// ---- DUTs/IO/Boxes/ER1008_78E8D3DD.TcDUT
{attribute 'GeneratedUsingTerminal: ER1008-0001-0016'}
{attribute addProperty BoxType "ER1008-0001-0016"}
{attribute addProperty Description "ER1008-0001 8 Ch. Dig. Input 24V, 3ms, M8"}
{attribute addProperty Physics "YY"}
{attribute addProperty Id "Channel_1AT %I*Channel_830843C11Channel_2AT %I*Channel_830843C11Channel_3AT %I*Channel_830843C11Channel_4AT %I*Channel_830843C11Channel_5AT %I*Channel_830843C11Channel_6AT %I*Channel_830843C11Channel_7AT %I*Channel_830843C11Channel_8AT %I*Channel_830843C11WcStateAT %I*WcState_9091E0EB2InfoDataAT %I*InfoData_6F19DB2B2"}
{attribute addProperty CRC "2028524509"}
{attribute addProperty Size "12"}
TYPE ER1008_78E8D3DD EXTENDS EtcSlaveBoxBase_77A0E4A7 :
STRUCT
	{attribute addProperty Name "Channel_1"}
	Channel_1 : Channel_830843C1;
	{attribute addProperty Name "Channel_2"}
	Channel_2 : Channel_830843C1;
	{attribute addProperty Name "Channel_3"}
	Channel_3 : Channel_830843C1;
	{attribute addProperty Name "Channel_4"}
	Channel_4 : Channel_830843C1;
	{attribute addProperty Name "Channel_5"}
	Channel_5 : Channel_830843C1;
	{attribute addProperty Name "Channel_6"}
	Channel_6 : Channel_830843C1;
	{attribute addProperty Name "Channel_7"}
	Channel_7 : Channel_830843C1;
	{attribute addProperty Name "Channel_8"}
	Channel_8 : Channel_830843C1;
	{attribute addProperty Name "WcState"}
	WcState : WcState_9091E0EB;
	{attribute addProperty Name "InfoData"}
	InfoData : InfoData_6F19DB2B;
END_STRUCT
END_TYPE

// ---- DUTs/IO/Boxes/ER1018_78E8D3DD.TcDUT
{attribute 'GeneratedUsingTerminal: ER1018-0001-0018'}
{attribute addProperty BoxType "ER1018-0001-0018"}
{attribute addProperty Description "ER1018-0001 8 Ch. Dig. Input 24V, 10µs, M8"}
{attribute addProperty Physics "YY"}
{attribute addProperty Id "Channel_1AT %I*Channel_830843C11Channel_2AT %I*Channel_830843C11Channel_3AT %I*Channel_830843C11Channel_4AT %I*Channel_830843C11Channel_5AT %I*Channel_830843C11Channel_6AT %I*Channel_830843C11Channel_7AT %I*Channel_830843C11Channel_8AT %I*Channel_830843C11WcStateAT %I*WcState_9091E0EB2InfoDataAT %I*InfoData_6F19DB2B2"}
{attribute addProperty CRC "2028524509"}
{attribute addProperty Size "12"}
TYPE ER1018_78E8D3DD EXTENDS EtcSlaveBoxBase_77A0E4A7 :
STRUCT
	{attribute addProperty Name "Channel_1"}
	Channel_1 : Channel_830843C1;
	{attribute addProperty Name "Channel_2"}
	Channel_2 : Channel_830843C1;
	{attribute addProperty Name "Channel_3"}
	Channel_3 : Channel_830843C1;
	{attribute addProperty Name "Channel_4"}
	Channel_4 : Channel_830843C1;
	{attribute addProperty Name "Channel_5"}
	Channel_5 : Channel_830843C1;
	{attribute addProperty Name "Channel_6"}
	Channel_6 : Channel_830843C1;
	{attribute addProperty Name "Channel_7"}
	Channel_7 : Channel_830843C1;
	{attribute addProperty Name "Channel_8"}
	Channel_8 : Channel_830843C1;
	{attribute addProperty Name "WcState"}
	WcState : WcState_9091E0EB;
	{attribute addProperty Name "InfoData"}
	InfoData : InfoData_6F19DB2B;
END_STRUCT
END_TYPE

// ---- DUTs/IO/Boxes/ER1098_78E8D3DD.TcDUT
{attribute 'GeneratedUsingTerminal: ER1098-0001-0017'}
{attribute addProperty BoxType "ER1098-0001-0017"}
{attribute addProperty Description "ER1098-0001 8 Ch. Dig. Input 24V, 10us, M8, negative"}
{attribute addProperty Physics "YY"}
{attribute addProperty Id "Channel_1AT %I*Channel_830843C11Channel_2AT %I*Channel_830843C11Channel_3AT %I*Channel_830843C11Channel_4AT %I*Channel_830843C11Channel_5AT %I*Channel_830843C11Channel_6AT %I*Channel_830843C11Channel_7AT %I*Channel_830843C11Channel_8AT %I*Channel_830843C11WcStateAT %I*WcState_9091E0EB2InfoDataAT %I*InfoData_6F19DB2B2"}
{attribute addProperty CRC "2028524509"}
{attribute addProperty Size "12"}
TYPE ER1098_78E8D3DD EXTENDS EtcSlaveBoxBase_77A0E4A7 :
STRUCT
	{attribute addProperty Name "Channel_1"}
	Channel_1 : Channel_830843C1;
	{attribute addProperty Name "Channel_2"}
	Channel_2 : Channel_830843C1;
	{attribute addProperty Name "Channel_3"}
	Channel_3 : Channel_830843C1;
	{attribute addProperty Name "Channel_4"}
	Channel_4 : Channel_830843C1;
	{attribute addProperty Name "Channel_5"}
	Channel_5 : Channel_830843C1;
	{attribute addProperty Name "Channel_6"}
	Channel_6 : Channel_830843C1;
	{attribute addProperty Name "Channel_7"}
	Channel_7 : Channel_830843C1;
	{attribute addProperty Name "Channel_8"}
	Channel_8 : Channel_830843C1;
	{attribute addProperty Name "WcState"}
	WcState : WcState_9091E0EB;
	{attribute addProperty Name "InfoData"}
	InfoData : InfoData_6F19DB2B;
END_STRUCT
END_TYPE

// ---- DUTs/IO/Boxes/ER1258_58F475DD.TcDUT
{attribute 'GeneratedUsingTerminal: ER1258-0001-0019'}
{attribute addProperty BoxType "ER1258-0001-0019"}
{attribute addProperty Description "ER1258-0001 8 Ch. Dig. Input 24V, 10µs, DC Latch, M8"}
{attribute addProperty Physics "YY"}
{attribute addProperty Id "Channel_1AT %I*Channel_830843C11Channel_2AT %I*Channel_830843C11Channel_3AT %I*Channel_830843C11Channel_4AT %I*Channel_830843C11Channel_5AT %I*Channel_830843C11Channel_6AT %I*Channel_830843C11Channel_7AT %I*Channel_830843C11Channel_8AT %I*Channel_830843C11LatchAT %I*Latch_8E41329534WcStateAT %I*WcState_B516A2644InfoDataAT %I*InfoData_A7436BC610"}
{attribute addProperty CRC "1492415965"}
{attribute addProperty Size "56"}
TYPE ER1258_58F475DD EXTENDS EtcSlaveBoxBase_77A0E4A7 :
STRUCT
	{attribute addProperty Name "Channel_1"}
	Channel_1 : Channel_830843C1;
	{attribute addProperty Name "Channel_2"}
	Channel_2 : Channel_830843C1;
	{attribute addProperty Name "Channel_3"}
	Channel_3 : Channel_830843C1;
	{attribute addProperty Name "Channel_4"}
	Channel_4 : Channel_830843C1;
	{attribute addProperty Name "Channel_5"}
	Channel_5 : Channel_830843C1;
	{attribute addProperty Name "Channel_6"}
	Channel_6 : Channel_830843C1;
	{attribute addProperty Name "Channel_7"}
	Channel_7 : Channel_830843C1;
	{attribute addProperty Name "Channel_8"}
	Channel_8 : Channel_830843C1;
	{attribute addProperty Name "Latch"}
	Latch : Latch_8E413295;
	{attribute addProperty Name "WcState"}
	WcState : WcState_B516A264;
	{attribute addProperty Name "InfoData"}
	InfoData : InfoData_A7436BC6;
END_STRUCT
END_TYPE

// ---- DUTs/IO/Boxes/ER1518_CC442588.TcDUT
{attribute 'GeneratedUsingTerminal: ER1518-0002-0018'}
{attribute addProperty BoxType "ER1518-0002-0018"}
{attribute addProperty Description "ER1518-0002 8 Ch.digital multi-function input"}
{attribute addProperty Physics "YY"}
{attribute addProperty Id "CNT_Input_Channel_1AT %I*CNT_Input_Channel_FF10BD3C11CNT_Input_Channel_2AT %I*CNT_Input_Channel_FF10BD3C11DIG_InputsAT %I*DIG_Inputs_CAFF60048DIG_Inputs_DeviceAT %I*DIG_Inputs_Device_1F4E72EB5CNT_Output_Channel_1AT %Q*CNT_Output_Channel_550BB6DF6CNT_Output_Channel_2AT %Q*CNT_Output_Channel_550BB6DF6WcStateAT %I*WcState_9091E0EB2InfoDataAT %I*InfoData_32EB74EA10"}
{attribute addProperty CRC "3427018120"}
{attribute addProperty Size "59"}
TYPE ER1518_CC442588 EXTENDS EtcSlaveBoxBase_77A0E4A7 :
STRUCT
	{attribute addProperty Name "CNT_Input_Channel_1"}
	CNT_Input_Channel_1 : CNT_Input_Channel_FF10BD3C;
	{attribute addProperty Name "CNT_Input_Channel_2"}
	CNT_Input_Channel_2 : CNT_Input_Channel_FF10BD3C;
	{attribute addProperty Name "DIG_Inputs"}
	DIG_Inputs : DIG_Inputs_CAFF6004;
	{attribute addProperty Name "DIG_Inputs_Device"}
	DIG_Inputs_Device : DIG_Inputs_Device_1F4E72EB;
	{attribute addProperty Name "CNT_Output_Channel_1"}
	CNT_Output_Channel_1 : CNT_Output_Channel_550BB6DF;
	{attribute addProperty Name "CNT_Output_Channel_2"}
	CNT_Output_Channel_2 : CNT_Output_Channel_550BB6DF;
	{attribute addProperty Name "WcState"}
	WcState : WcState_9091E0EB;
	{attribute addProperty Name "InfoData"}
	InfoData : InfoData_32EB74EA;
END_STRUCT
END_TYPE

// ---- DUTs/IO/Boxes/ER1809_32157CFD.TcDUT
{attribute 'GeneratedUsingTerminal: ER1809-0021-0017'}
{attribute addProperty BoxType "ER1809-0021-0017"}
{attribute addProperty Description "ER1809-0021 16 Ch. Dig. Input 24V, 3ms, M8"}
{attribute addProperty Physics "YY"}
{attribute addProperty Id "Channel_1AT %I*Channel_830843C11Channel_2AT %I*Channel_830843C11Channel_3AT %I*Channel_830843C11Channel_4AT %I*Channel_830843C11Channel_5AT %I*Channel_830843C11Channel_6AT %I*Channel_830843C11Channel_7AT %I*Channel_830843C11Channel_8AT %I*Channel_830843C11Channel_9AT %I*Channel_830843C11Channel_10AT %I*Channel_830843C11Channel_11AT %I*Channel_830843C11Channel_12AT %I*Channel_830843C11Channel_13AT %I*Channel_830843C11Channel_14AT %I*Channel_830843C11Channel_15AT %I*Channel_830843C11Channel_16AT %I*Channel_830843C11WcStateAT %I*WcState_9091E0EB2InfoDataAT %I*InfoData_6F19DB2B2"}
{attribute addProperty CRC "840269053"}
{attribute addProperty Size "20"}
TYPE ER1809_32157CFD EXTENDS EtcSlaveBoxBase_77A0E4A7 :
STRUCT
	{attribute addProperty Name "Channel_1"}
	Channel_1 : Channel_830843C1;
	{attribute addProperty Name "Channel_2"}
	Channel_2 : Channel_830843C1;
	{attribute addProperty Name "Channel_3"}
	Channel_3 : Channel_830843C1;
	{attribute addProperty Name "Channel_4"}
	Channel_4 : Channel_830843C1;
	{attribute addProperty Name "Channel_5"}
	Channel_5 : Channel_830843C1;
	{attribute addProperty Name "Channel_6"}
	Channel_6 : Channel_830843C1;
	{attribute addProperty Name "Channel_7"}
	Channel_7 : Channel_830843C1;
	{attribute addProperty Name "Channel_8"}
	Channel_8 : Channel_830843C1;
	{attribute addProperty Name "Channel_9"}
	Channel_9 : Channel_830843C1;
	{attribute addProperty Name "Channel_10"}
	Channel_10 : Channel_830843C1;
	{attribute addProperty Name "Channel_11"}
	Channel_11 : Channel_830843C1;
	{attribute addProperty Name "Channel_12"}
	Channel_12 : Channel_830843C1;
	{attribute addProperty Name "Channel_13"}
	Channel_13 : Channel_830843C1;
	{attribute addProperty Name "Channel_14"}
	Channel_14 : Channel_830843C1;
	{attribute addProperty Name "Channel_15"}
	Channel_15 : Channel_830843C1;
	{attribute addProperty Name "Channel_16"}
	Channel_16 : Channel_830843C1;
	{attribute addProperty Name "WcState"}
	WcState : WcState_9091E0EB;
	{attribute addProperty Name "InfoData"}
	InfoData : InfoData_6F19DB2B;
END_STRUCT
END_TYPE

// ---- DUTs/IO/Boxes/ER1819_32157CFD.TcDUT
{attribute 'GeneratedUsingTerminal: ER1819-0021-0017'}
{attribute addProperty BoxType "ER1819-0021-0017"}
{attribute addProperty Description "ER1819-0021 16 Ch. Dig. Input 24V, 10µs, M8"}
{attribute addProperty Physics "YY"}
{attribute addProperty Id "Channel_1AT %I*Channel_830843C11Channel_2AT %I*Channel_830843C11Channel_3AT %I*Channel_830843C11Channel_4AT %I*Channel_830843C11Channel_5AT %I*Channel_830843C11Channel_6AT %I*Channel_830843C11Channel_7AT %I*Channel_830843C11Channel_8AT %I*Channel_830843C11Channel_9AT %I*Channel_830843C11Channel_10AT %I*Channel_830843C11Channel_11AT %I*Channel_830843C11Channel_12AT %I*Channel_830843C11Channel_13AT %I*Channel_830843C11Channel_14AT %I*Channel_830843C11Channel_15AT %I*Channel_830843C11Channel_16AT %I*Channel_830843C11WcStateAT %I*WcState_9091E0EB2InfoDataAT %I*InfoData_6F19DB2B2"}
{attribute addProperty CRC "840269053"}
{attribute addProperty Size "20"}
TYPE ER1819_32157CFD EXTENDS EtcSlaveBoxBase_77A0E4A7 :
STRUCT
	{attribute addProperty Name "Channel_1"}
	Channel_1 : Channel_830843C1;
	{attribute addProperty Name "Channel_2"}
	Channel_2 : Channel_830843C1;
	{attribute addProperty Name "Channel_3"}
	Channel_3 : Channel_830843C1;
	{attribute addProperty Name "Channel_4"}
	Channel_4 : Channel_830843C1;
	{attribute addProperty Name "Channel_5"}
	Channel_5 : Channel_830843C1;
	{attribute addProperty Name "Channel_6"}
	Channel_6 : Channel_830843C1;
	{attribute addProperty Name "Channel_7"}
	Channel_7 : Channel_830843C1;
	{attribute addProperty Name "Channel_8"}
	Channel_8 : Channel_830843C1;
	{attribute addProperty Name "Channel_9"}
	Channel_9 : Channel_830843C1;
	{attribute addProperty Name "Channel_10"}
	Channel_10 : Channel_830843C1;
	{attribute addProperty Name "Channel_11"}
	Channel_11 : Channel_830843C1;
	{attribute addProperty Name "Channel_12"}
	Channel_12 : Channel_830843C1;
	{attribute addProperty Name "Channel_13"}
	Channel_13 : Channel_830843C1;
	{attribute addProperty Name "Channel_14"}
	Channel_14 : Channel_830843C1;
	{attribute addProperty Name "Channel_15"}
	Channel_15 : Channel_830843C1;
	{attribute addProperty Name "Channel_16"}
	Channel_16 : Channel_830843C1;
	{attribute addProperty Name "WcState"}
	WcState : WcState_9091E0EB;
	{attribute addProperty Name "InfoData"}
	InfoData : InfoData_6F19DB2B;
END_STRUCT
END_TYPE

// ---- DUTs/IO/Boxes/ER2008_E2806B95.TcDUT
{attribute 'GeneratedUsingTerminal: ER2008-0001-0018'}
{attribute addProperty BoxType "ER2008-0001-0018"}
{attribute addProperty Description "ER2008-0001 8 Ch. Dig. Output 24V, 0,5A, M8"}
{attribute addProperty Physics "YY"}
{attribute addProperty Id "Channel_1AT %Q*Channel_42CA91F71Channel_2AT %Q*Channel_42CA91F71Channel_3AT %Q*Channel_42CA91F71Channel_4AT %Q*Channel_42CA91F71Channel_5AT %Q*Channel_42CA91F71Channel_6AT %Q*Channel_42CA91F71Channel_7AT %Q*Channel_42CA91F71Channel_8AT %Q*Channel_42CA91F71WcStateAT %I*WcState_0B2B16F91InfoDataAT %I*InfoData_6F19DB2B2"}
{attribute addProperty CRC "3800066965"}
{attribute addProperty Size "11"}
TYPE ER2008_E2806B95 EXTENDS EtcSlaveBoxBase_77A0E4A7 :
STRUCT
	{attribute addProperty Name "Channel_1"}
	Channel_1 : Channel_42CA91F7;
	{attribute addProperty Name "Channel_2"}
	Channel_2 : Channel_42CA91F7;
	{attribute addProperty Name "Channel_3"}
	Channel_3 : Channel_42CA91F7;
	{attribute addProperty Name "Channel_4"}
	Channel_4 : Channel_42CA91F7;
	{attribute addProperty Name "Channel_5"}
	Channel_5 : Channel_42CA91F7;
	{attribute addProperty Name "Channel_6"}
	Channel_6 : Channel_42CA91F7;
	{attribute addProperty Name "Channel_7"}
	Channel_7 : Channel_42CA91F7;
	{attribute addProperty Name "Channel_8"}
	Channel_8 : Channel_42CA91F7;
	{attribute addProperty Name "WcState"}
	WcState : WcState_0B2B16F9;
	{attribute addProperty Name "InfoData"}
	InfoData : InfoData_6F19DB2B;
END_STRUCT
END_TYPE

// ---- DUTs/IO/Boxes/ER2028_E2806B95.TcDUT
{attribute 'GeneratedUsingTerminal: ER2028-0001-0017'}
{attribute addProperty BoxType "ER2028-0001-0017"}
{attribute addProperty Description "ER2028-0001 8 Ch. Dig. Output 24V, 2A, M8"}
{attribute addProperty Physics "YY"}
{attribute addProperty Id "Channel_1AT %Q*Channel_42CA91F71Channel_2AT %Q*Channel_42CA91F71Channel_3AT %Q*Channel_42CA91F71Channel_4AT %Q*Channel_42CA91F71Channel_5AT %Q*Channel_42CA91F71Channel_6AT %Q*Channel_42CA91F71Channel_7AT %Q*Channel_42CA91F71Channel_8AT %Q*Channel_42CA91F71WcStateAT %I*WcState_0B2B16F91InfoDataAT %I*InfoData_6F19DB2B2"}
{attribute addProperty CRC "3800066965"}
{attribute addProperty Size "11"}
TYPE ER2028_E2806B95 EXTENDS EtcSlaveBoxBase_77A0E4A7 :
STRUCT
	{attribute addProperty Name "Channel_1"}
	Channel_1 : Channel_42CA91F7;
	{attribute addProperty Name "Channel_2"}
	Channel_2 : Channel_42CA91F7;
	{attribute addProperty Name "Channel_3"}
	Channel_3 : Channel_42CA91F7;
	{attribute addProperty Name "Channel_4"}
	Channel_4 : Channel_42CA91F7;
	{attribute addProperty Name "Channel_5"}
	Channel_5 : Channel_42CA91F7;
	{attribute addProperty Name "Channel_6"}
	Channel_6 : Channel_42CA91F7;
	{attribute addProperty Name "Channel_7"}
	Channel_7 : Channel_42CA91F7;
	{attribute addProperty Name "Channel_8"}
	Channel_8 : Channel_42CA91F7;
	{attribute addProperty Name "WcState"}
	WcState : WcState_0B2B16F9;
	{attribute addProperty Name "InfoData"}
	InfoData : InfoData_6F19DB2B;
END_STRUCT
END_TYPE

// ---- DUTs/IO/Boxes/ER2038_3AE10DD7.TcDUT
{attribute 'GeneratedUsingTerminal: ER2038-0001-0017'}
{attribute addProperty BoxType "ER2038-0001-0017"}
{attribute addProperty Description "ER2038-0001 8 Ch. Dig. Output 24V, 2A, M8, Diagnostic"}
{attribute addProperty Physics "YY"}
{attribute addProperty Id "Diag_Channel_1AT %I*Diag_Channel_830843C11Diag_Channel_2AT %I*Diag_Channel_830843C11Diag_Channel_3AT %I*Diag_Channel_830843C11Diag_Channel_4AT %I*Diag_Channel_830843C11Diag_Channel_5AT %I*Diag_Channel_830843C11Diag_Channel_6AT %I*Diag_Channel_830843C11Diag_Channel_7AT %I*Diag_Channel_830843C11Diag_Channel_8AT %I*Diag_Channel_830843C11Channel_1AT %Q*Channel_42CA91F71Channel_2AT %Q*Channel_42CA91F71Channel_3AT %Q*Channel_42CA91F71Channel_4AT %Q*Channel_42CA91F71Channel_5AT %Q*Channel_42CA91F71Channel_6AT %Q*Channel_42CA91F71Channel_7AT %Q*Channel_42CA91F71Channel_8AT %Q*Channel_42CA91F71WcStateAT %I*WcState_9091E0EB2InfoDataAT %I*InfoData_6F19DB2B2"}
{attribute addProperty CRC "987827671"}
{attribute addProperty Size "20"}
TYPE ER2038_3AE10DD7 EXTENDS EtcSlaveBoxBase_77A0E4A7 :
STRUCT
	{attribute addProperty Name "Diag_Channel_1"}
	Diag_Channel_1 : Diag_Channel_830843C1;
	{attribute addProperty Name "Diag_Channel_2"}
	Diag_Channel_2 : Diag_Channel_830843C1;
	{attribute addProperty Name "Diag_Channel_3"}
	Diag_Channel_3 : Diag_Channel_830843C1;
	{attribute addProperty Name "Diag_Channel_4"}
	Diag_Channel_4 : Diag_Channel_830843C1;
	{attribute addProperty Name "Diag_Channel_5"}
	Diag_Channel_5 : Diag_Channel_830843C1;
	{attribute addProperty Name "Diag_Channel_6"}
	Diag_Channel_6 : Diag_Channel_830843C1;
	{attribute addProperty Name "Diag_Channel_7"}
	Diag_Channel_7 : Diag_Channel_830843C1;
	{attribute addProperty Name "Diag_Channel_8"}
	Diag_Channel_8 : Diag_Channel_830843C1;
	{attribute addProperty Name "Channel_1"}
	Channel_1 : Channel_42CA91F7;
	{attribute addProperty Name "Channel_2"}
	Channel_2 : Channel_42CA91F7;
	{attribute addProperty Name "Channel_3"}
	Channel_3 : Channel_42CA91F7;
	{attribute addProperty Name "Channel_4"}
	Channel_4 : Channel_42CA91F7;
	{attribute addProperty Name "Channel_5"}
	Channel_5 : Channel_42CA91F7;
	{attribute addProperty Name "Channel_6"}
	Channel_6 : Channel_42CA91F7;
	{attribute addProperty Name "Channel_7"}
	Channel_7 : Channel_42CA91F7;
	{attribute addProperty Name "Channel_8"}
	Channel_8 : Channel_42CA91F7;
	{attribute addProperty Name "WcState"}
	WcState : WcState_9091E0EB;
	{attribute addProperty Name "InfoData"}
	InfoData : InfoData_6F19DB2B;
END_STRUCT
END_TYPE

// ---- DUTs/IO/Boxes/ER2308_F6D9A8D1.TcDUT
{attribute 'GeneratedUsingTerminal: ER2308-0001-0018'}
{attribute addProperty BoxType "ER2308-0001-0018"}
{attribute addProperty Description "ER2308-0001 4 Ch. Dig. In, 3ms, 4 Ch. Dig. Out 24V, 0,5A, M8"}
{attribute addProperty Physics "YY"}
{attribute addProperty Id "Channel_1AT %I*Channel_830843C11Channel_2AT %I*Channel_830843C11Channel_3AT %I*Channel_830843C11Channel_4AT %I*Channel_830843C11Channel_5AT %Q*Channel_42CA91F71Channel_6AT %Q*Channel_42CA91F71Channel_7AT %Q*Channel_42CA91F71Channel_8AT %Q*Channel_42CA91F71WcStateAT %I*WcState_9091E0EB2InfoDataAT %I*InfoData_6F19DB2B2"}
{attribute addProperty CRC "4141459665"}
{attribute addProperty Size "12"}
TYPE ER2308_F6D9A8D1 EXTENDS EtcSlaveBoxBase_77A0E4A7 :
STRUCT
	{attribute addProperty Name "Channel_1"}
	Channel_1 : Channel_830843C1;
	{attribute addProperty Name "Channel_2"}
	Channel_2 : Channel_830843C1;
	{attribute addProperty Name "Channel_3"}
	Channel_3 : Channel_830843C1;
	{attribute addProperty Name "Channel_4"}
	Channel_4 : Channel_830843C1;
	{attribute addProperty Name "Channel_5"}
	Channel_5 : Channel_42CA91F7;
	{attribute addProperty Name "Channel_6"}
	Channel_6 : Channel_42CA91F7;
	{attribute addProperty Name "Channel_7"}
	Channel_7 : Channel_42CA91F7;
	{attribute addProperty Name "Channel_8"}
	Channel_8 : Channel_42CA91F7;
	{attribute addProperty Name "WcState"}
	WcState : WcState_9091E0EB;
	{attribute addProperty Name "InfoData"}
	InfoData : InfoData_6F19DB2B;
END_STRUCT
END_TYPE

// ---- DUTs/IO/Boxes/ER2318_F6D9A8D1.TcDUT
{attribute 'GeneratedUsingTerminal: ER2318-0001-0018'}
{attribute addProperty BoxType "ER2318-0001-0018"}
{attribute addProperty Description "ER2318-0001 4 Ch. Dig. In, 10µs, 4 Ch. Dig. Out 24V, 0,5A, M8"}
{attribute addProperty Physics "YY"}
{attribute addProperty Id "Channel_1AT %I*Channel_830843C11Channel_2AT %I*Channel_830843C11Channel_3AT %I*Channel_830843C11Channel_4AT %I*Channel_830843C11Channel_5AT %Q*Channel_42CA91F71Channel_6AT %Q*Channel_42CA91F71Channel_7AT %Q*Channel_42CA91F71Channel_8AT %Q*Channel_42CA91F71WcStateAT %I*WcState_9091E0EB2InfoDataAT %I*InfoData_6F19DB2B2"}
{attribute addProperty CRC "4141459665"}
{attribute addProperty Size "12"}
TYPE ER2318_F6D9A8D1 EXTENDS EtcSlaveBoxBase_77A0E4A7 :
STRUCT
	{attribute addProperty Name "Channel_1"}
	Channel_1 : Channel_830843C1;
	{attribute addProperty Name "Channel_2"}
	Channel_2 : Channel_830843C1;
	{attribute addProperty Name "Channel_3"}
	Channel_3 : Channel_830843C1;
	{attribute addProperty Name "Channel_4"}
	Channel_4 : Channel_830843C1;
	{attribute addProperty Name "Channel_5"}
	Channel_5 : Channel_42CA91F7;
	{attribute addProperty Name "Channel_6"}
	Channel_6 : Channel_42CA91F7;
	{attribute addProperty Name "Channel_7"}
	Channel_7 : Channel_42CA91F7;
	{attribute addProperty Name "Channel_8"}
	Channel_8 : Channel_42CA91F7;
	{attribute addProperty Name "WcState"}
	WcState : WcState_9091E0EB;
	{attribute addProperty Name "InfoData"}
	InfoData : InfoData_6F19DB2B;
END_STRUCT
END_TYPE

// ---- DUTs/IO/Boxes/ER2328_F6D9A8D1.TcDUT
{attribute 'GeneratedUsingTerminal: ER2328-0001-0017'}
{attribute addProperty BoxType "ER2328-0001-0017"}
{attribute addProperty Description "ER2328-0001 4 CH. Dig. In, 3ms, 4 Ch. Dig. Out 24V, 2A, M8"}
{attribute addProperty Physics "YY"}
{attribute addProperty Id "Channel_1AT %I*Channel_830843C11Channel_2AT %I*Channel_830843C11Channel_3AT %I*Channel_830843C11Channel_4AT %I*Channel_830843C11Channel_5AT %Q*Channel_42CA91F71Channel_6AT %Q*Channel_42CA91F71Channel_7AT %Q*Channel_42CA91F71Channel_8AT %Q*Channel_42CA91F71WcStateAT %I*WcState_9091E0EB2InfoDataAT %I*InfoData_6F19DB2B2"}
{attribute addProperty CRC "4141459665"}
{attribute addProperty Size "12"}
TYPE ER2328_F6D9A8D1 EXTENDS EtcSlaveBoxBase_77A0E4A7 :
STRUCT
	{attribute addProperty Name "Channel_1"}
	Channel_1 : Channel_830843C1;
	{attribute addProperty Name "Channel_2"}
	Channel_2 : Channel_830843C1;
	{attribute addProperty Name "Channel_3"}
	Channel_3 : Channel_830843C1;
	{attribute addProperty Name "Channel_4"}
	Channel_4 : Channel_830843C1;
	{attribute addProperty Name "Channel_5"}
	Channel_5 : Channel_42CA91F7;
	{attribute addProperty Name "Channel_6"}
	Channel_6 : Channel_42CA91F7;
	{attribute addProperty Name "Channel_7"}
	Channel_7 : Channel_42CA91F7;
	{attribute addProperty Name "Channel_8"}
	Channel_8 : Channel_42CA91F7;
	{attribute addProperty Name "WcState"}
	WcState : WcState_9091E0EB;
	{attribute addProperty Name "InfoData"}
	InfoData : InfoData_6F19DB2B;
END_STRUCT
END_TYPE

// ---- DUTs/IO/Boxes/ER2338_7699BCF6.TcDUT
{attribute 'GeneratedUsingTerminal: ER2338-0001-0022'}
{attribute addProperty BoxType "ER2338-0001-0022"}
{attribute addProperty Description "ER2338-0001 8 Ch. Dig. Input/Output 24V, 0,5A, M8"}
{attribute addProperty Physics "YY"}
{attribute addProperty Id "Channel_1AT %I*Channel_830843C11Channel_2AT %I*Channel_830843C11Channel_3AT %I*Channel_830843C11Channel_4AT %I*Channel_830843C11Channel_5AT %I*Channel_830843C11Channel_6AT %I*Channel_830843C11Channel_7AT %I*Channel_830843C11Channel_8AT %I*Channel_830843C11Channel_9AT %Q*Channel_42CA91F71Channel_10AT %Q*Channel_42CA91F71Channel_11AT %Q*Channel_42CA91F71Channel_12AT %Q*Channel_42CA91F71Channel_13AT %Q*Channel_42CA91F71Channel_14AT %Q*Channel_42CA91F71Channel_15AT %Q*Channel_42CA91F71Channel_16AT %Q*Channel_42CA91F71WcStateAT %I*WcState_9091E0EB2InfoDataAT %I*InfoData_6F19DB2B2"}
{attribute addProperty CRC "1989786870"}
{attribute addProperty Size "20"}
TYPE ER2338_7699BCF6 EXTENDS EtcSlaveBoxBase_77A0E4A7 :
STRUCT
	{attribute addProperty Name "Channel_1"}
	Channel_1 : Channel_830843C1;
	{attribute addProperty Name "Channel_2"}
	Channel_2 : Channel_830843C1;
	{attribute addProperty Name "Channel_3"}
	Channel_3 : Channel_830843C1;
	{attribute addProperty Name "Channel_4"}
	Channel_4 : Channel_830843C1;
	{attribute addProperty Name "Channel_5"}
	Channel_5 : Channel_830843C1;
	{attribute addProperty Name "Channel_6"}
	Channel_6 : Channel_830843C1;
	{attribute addProperty Name "Channel_7"}
	Channel_7 : Channel_830843C1;
	{attribute addProperty Name "Channel_8"}
	Channel_8 : Channel_830843C1;
	{attribute addProperty Name "Channel_9"}
	Channel_9 : Channel_42CA91F7;
	{attribute addProperty Name "Channel_10"}
	Channel_10 : Channel_42CA91F7;
	{attribute addProperty Name "Channel_11"}
	Channel_11 : Channel_42CA91F7;
	{attribute addProperty Name "Channel_12"}
	Channel_12 : Channel_42CA91F7;
	{attribute addProperty Name "Channel_13"}
	Channel_13 : Channel_42CA91F7;
	{attribute addProperty Name "Channel_14"}
	Channel_14 : Channel_42CA91F7;
	{attribute addProperty Name "Channel_15"}
	Channel_15 : Channel_42CA91F7;
	{attribute addProperty Name "Channel_16"}
	Channel_16 : Channel_42CA91F7;
	{attribute addProperty Name "WcState"}
	WcState : WcState_9091E0EB;
	{attribute addProperty Name "InfoData"}
	InfoData : InfoData_6F19DB2B;
END_STRUCT
END_TYPE

// ---- DUTs/IO/Boxes/ER2339_D8E9F29A.TcDUT
{attribute 'GeneratedUsingTerminal: ER2339-0021-0018'}
{attribute addProperty BoxType "ER2339-0021-0018"}
{attribute addProperty Description "ER2339-0021 16 Ch. Dig. Input/Output 24V, 0,5A, M8"}
{attribute addProperty Physics "YY"}
{attribute addProperty Id "Channel_1AT %I*Channel_830843C11Channel_2AT %I*Channel_830843C11Channel_3AT %I*Channel_830843C11Channel_4AT %I*Channel_830843C11Channel_5AT %I*Channel_830843C11Channel_6AT %I*Channel_830843C11Channel_7AT %I*Channel_830843C11Channel_8AT %I*Channel_830843C11Channel_9AT %I*Channel_830843C11Channel_10AT %I*Channel_830843C11Channel_11AT %I*Channel_830843C11Channel_12AT %I*Channel_830843C11Channel_13AT %I*Channel_830843C11Channel_14AT %I*Channel_830843C11Channel_15AT %I*Channel_830843C11Channel_16AT %I*Channel_830843C11Channel_17AT %Q*Channel_42CA91F71Channel_18AT %Q*Channel_42CA91F71Channel_19AT %Q*Channel_42CA91F71Channel_20AT %Q*Channel_42CA91F71Channel_21AT %Q*Channel_42CA91F71Channel_22AT %Q*Channel_42CA91F71Channel_23AT %Q*Channel_42CA91F71Channel_24AT %Q*Channel_42CA91F71Channel_25AT %Q*Channel_42CA91F71Channel_26AT %Q*Channel_42CA91F71Channel_27AT %Q*Channel_42CA91F71Channel_28AT %Q*Channel_42CA91F71Channel_29AT %Q*Channel_42CA91F71Channel_30AT %Q*Channel_42CA91F71Channel_31AT %Q*Channel_42CA91F71Channel_32AT %Q*Channel_42CA91F71WcStateAT %I*WcState_9091E0EB2InfoDataAT %I*InfoData_0A66F0098"}
{attribute addProperty CRC "3639210650"}
{attribute addProperty Size "42"}
TYPE ER2339_D8E9F29A EXTENDS EtcSlaveBoxBase_77A0E4A7 :
STRUCT
	{attribute addProperty Name "Channel_1"}
	Channel_1 : Channel_830843C1;
	{attribute addProperty Name "Channel_2"}
	Channel_2 : Channel_830843C1;
	{attribute addProperty Name "Channel_3"}
	Channel_3 : Channel_830843C1;
	{attribute addProperty Name "Channel_4"}
	Channel_4 : Channel_830843C1;
	{attribute addProperty Name "Channel_5"}
	Channel_5 : Channel_830843C1;
	{attribute addProperty Name "Channel_6"}
	Channel_6 : Channel_830843C1;
	{attribute addProperty Name "Channel_7"}
	Channel_7 : Channel_830843C1;
	{attribute addProperty Name "Channel_8"}
	Channel_8 : Channel_830843C1;
	{attribute addProperty Name "Channel_9"}
	Channel_9 : Channel_830843C1;
	{attribute addProperty Name "Channel_10"}
	Channel_10 : Channel_830843C1;
	{attribute addProperty Name "Channel_11"}
	Channel_11 : Channel_830843C1;
	{attribute addProperty Name "Channel_12"}
	Channel_12 : Channel_830843C1;
	{attribute addProperty Name "Channel_13"}
	Channel_13 : Channel_830843C1;
	{attribute addProperty Name "Channel_14"}
	Channel_14 : Channel_830843C1;
	{attribute addProperty Name "Channel_15"}
	Channel_15 : Channel_830843C1;
	{attribute addProperty Name "Channel_16"}
	Channel_16 : Channel_830843C1;
	{attribute addProperty Name "Channel_17"}
	Channel_17 : Channel_42CA91F7;
	{attribute addProperty Name "Channel_18"}
	Channel_18 : Channel_42CA91F7;
	{attribute addProperty Name "Channel_19"}
	Channel_19 : Channel_42CA91F7;
	{attribute addProperty Name "Channel_20"}
	Channel_20 : Channel_42CA91F7;
	{attribute addProperty Name "Channel_21"}
	Channel_21 : Channel_42CA91F7;
	{attribute addProperty Name "Channel_22"}
	Channel_22 : Channel_42CA91F7;
	{attribute addProperty Name "Channel_23"}
	Channel_23 : Channel_42CA91F7;
	{attribute addProperty Name "Channel_24"}
	Channel_24 : Channel_42CA91F7;
	{attribute addProperty Name "Channel_25"}
	Channel_25 : Channel_42CA91F7;
	{attribute addProperty Name "Channel_26"}
	Channel_26 : Channel_42CA91F7;
	{attribute addProperty Name "Channel_27"}
	Channel_27 : Channel_42CA91F7;
	{attribute addProperty Name "Channel_28"}
	Channel_28 : Channel_42CA91F7;
	{attribute addProperty Name "Channel_29"}
	Channel_29 : Channel_42CA91F7;
	{attribute addProperty Name "Channel_30"}
	Channel_30 : Channel_42CA91F7;
	{attribute addProperty Name "Channel_31"}
	Channel_31 : Channel_42CA91F7;
	{attribute addProperty Name "Channel_32"}
	Channel_32 : Channel_42CA91F7;
	{attribute addProperty Name "WcState"}
	WcState : WcState_9091E0EB;
	{attribute addProperty Name "InfoData"}
	InfoData : InfoData_0A66F009;
END_STRUCT
END_TYPE

// ---- DUTs/IO/Boxes/ER2339_4CF33DED.TcDUT
{attribute 'GeneratedUsingTerminal: ER2339-0021-0019'}
{attribute addProperty BoxType "ER2339-0021-0019"}
{attribute addProperty Description "ER2339-0021 16 Ch. Dig. Input/Output 24V, 0,5A, M8"}
{attribute addProperty Physics "YY"}
{attribute addProperty Id "Channel_1AT %I*Channel_830843C11Channel_2AT %I*Channel_830843C11Channel_3AT %I*Channel_830843C11Channel_4AT %I*Channel_830843C11Channel_5AT %I*Channel_830843C11Channel_6AT %I*Channel_830843C11Channel_7AT %I*Channel_830843C11Channel_8AT %I*Channel_830843C11Channel_9AT %I*Channel_830843C11Channel_10AT %I*Channel_830843C11Channel_11AT %I*Channel_830843C11Channel_12AT %I*Channel_830843C11Channel_13AT %I*Channel_830843C11Channel_14AT %I*Channel_830843C11Channel_15AT %I*Channel_830843C11Channel_16AT %I*Channel_830843C11Channel_17AT %Q*Channel_42CA91F71Channel_18AT %Q*Channel_42CA91F71Channel_19AT %Q*Channel_42CA91F71Channel_20AT %Q*Channel_42CA91F71Channel_21AT %Q*Channel_42CA91F71Channel_22AT %Q*Channel_42CA91F71Channel_23AT %Q*Channel_42CA91F71Channel_24AT %Q*Channel_42CA91F71Channel_25AT %Q*Channel_42CA91F71Channel_26AT %Q*Channel_42CA91F71Channel_27AT %Q*Channel_42CA91F71Channel_28AT %Q*Channel_42CA91F71Channel_29AT %Q*Channel_42CA91F71Channel_30AT %Q*Channel_42CA91F71Channel_31AT %Q*Channel_42CA91F71Channel_32AT %Q*Channel_42CA91F71WcStateAT %I*WcState_9091E0EB2InfoDataAT %I*InfoData_6F19DB2B2"}
{attribute addProperty CRC "1291009517"}
{attribute addProperty Size "36"}
TYPE ER2339_4CF33DED EXTENDS EtcSlaveBoxBase_77A0E4A7 :
STRUCT
	{attribute addProperty Name "Channel_1"}
	Channel_1 : Channel_830843C1;
	{attribute addProperty Name "Channel_2"}
	Channel_2 : Channel_830843C1;
	{attribute addProperty Name "Channel_3"}
	Channel_3 : Channel_830843C1;
	{attribute addProperty Name "Channel_4"}
	Channel_4 : Channel_830843C1;
	{attribute addProperty Name "Channel_5"}
	Channel_5 : Channel_830843C1;
	{attribute addProperty Name "Channel_6"}
	Channel_6 : Channel_830843C1;
	{attribute addProperty Name "Channel_7"}
	Channel_7 : Channel_830843C1;
	{attribute addProperty Name "Channel_8"}
	Channel_8 : Channel_830843C1;
	{attribute addProperty Name "Channel_9"}
	Channel_9 : Channel_830843C1;
	{attribute addProperty Name "Channel_10"}
	Channel_10 : Channel_830843C1;
	{attribute addProperty Name "Channel_11"}
	Channel_11 : Channel_830843C1;
	{attribute addProperty Name "Channel_12"}
	Channel_12 : Channel_830843C1;
	{attribute addProperty Name "Channel_13"}
	Channel_13 : Channel_830843C1;
	{attribute addProperty Name "Channel_14"}
	Channel_14 : Channel_830843C1;
	{attribute addProperty Name "Channel_15"}
	Channel_15 : Channel_830843C1;
	{attribute addProperty Name "Channel_16"}
	Channel_16 : Channel_830843C1;
	{attribute addProperty Name "Channel_17"}
	Channel_17 : Channel_42CA91F7;
	{attribute addProperty Name "Channel_18"}
	Channel_18 : Channel_42CA91F7;
	{attribute addProperty Name "Channel_19"}
	Channel_19 : Channel_42CA91F7;
	{attribute addProperty Name "Channel_20"}
	Channel_20 : Channel_42CA91F7;
	{attribute addProperty Name "Channel_21"}
	Channel_21 : Channel_42CA91F7;
	{attribute addProperty Name "Channel_22"}
	Channel_22 : Channel_42CA91F7;
	{attribute addProperty Name "Channel_23"}
	Channel_23 : Channel_42CA91F7;
	{attribute addProperty Name "Channel_24"}
	Channel_24 : Channel_42CA91F7;
	{attribute addProperty Name "Channel_25"}
	Channel_25 : Channel_42CA91F7;
	{attribute addProperty Name "Channel_26"}
	Channel_26 : Channel_42CA91F7;
	{attribute addProperty Name "Channel_27"}
	Channel_27 : Channel_42CA91F7;
	{attribute addProperty Name "Channel_28"}
	Channel_28 : Channel_42CA91F7;
	{attribute addProperty Name "Channel_29"}
	Channel_29 : Channel_42CA91F7;
	{attribute addProperty Name "Channel_30"}
	Channel_30 : Channel_42CA91F7;
	{attribute addProperty Name "Channel_31"}
	Channel_31 : Channel_42CA91F7;
	{attribute addProperty Name "Channel_32"}
	Channel_32 : Channel_42CA91F7;
	{attribute addProperty Name "WcState"}
	WcState : WcState_9091E0EB;
	{attribute addProperty Name "InfoData"}
	InfoData : InfoData_6F19DB2B;
END_STRUCT
END_TYPE

// ---- DUTs/IO/Boxes/ER2349_4CF33DED.TcDUT
{attribute 'GeneratedUsingTerminal: ER2349-0021-0017'}
{attribute addProperty BoxType "ER2349-0021-0017"}
{attribute addProperty Description "ER2349-0021 16 Ch. Dig. Input/Output 24V, 10µs, 0,5A, M8"}
{attribute addProperty Physics "YY"}
{attribute addProperty Id "Channel_1AT %I*Channel_830843C11Channel_2AT %I*Channel_830843C11Channel_3AT %I*Channel_830843C11Channel_4AT %I*Channel_830843C11Channel_5AT %I*Channel_830843C11Channel_6AT %I*Channel_830843C11Channel_7AT %I*Channel_830843C11Channel_8AT %I*Channel_830843C11Channel_9AT %I*Channel_830843C11Channel_10AT %I*Channel_830843C11Channel_11AT %I*Channel_830843C11Channel_12AT %I*Channel_830843C11Channel_13AT %I*Channel_830843C11Channel_14AT %I*Channel_830843C11Channel_15AT %I*Channel_830843C11Channel_16AT %I*Channel_830843C11Channel_17AT %Q*Channel_42CA91F71Channel_18AT %Q*Channel_42CA91F71Channel_19AT %Q*Channel_42CA91F71Channel_20AT %Q*Channel_42CA91F71Channel_21AT %Q*Channel_42CA91F71Channel_22AT %Q*Channel_42CA91F71Channel_23AT %Q*Channel_42CA91F71Channel_24AT %Q*Channel_42CA91F71Channel_25AT %Q*Channel_42CA91F71Channel_26AT %Q*Channel_42CA91F71Channel_27AT %Q*Channel_42CA91F71Channel_28AT %Q*Channel_42CA91F71Channel_29AT %Q*Channel_42CA91F71Channel_30AT %Q*Channel_42CA91F71Channel_31AT %Q*Channel_42CA91F71Channel_32AT %Q*Channel_42CA91F71WcStateAT %I*WcState_9091E0EB2InfoDataAT %I*InfoData_6F19DB2B2"}
{attribute addProperty CRC "1291009517"}
{attribute addProperty Size "36"}
TYPE ER2349_4CF33DED EXTENDS EtcSlaveBoxBase_77A0E4A7 :
STRUCT
	{attribute addProperty Name "Channel_1"}
	Channel_1 : Channel_830843C1;
	{attribute addProperty Name "Channel_2"}
	Channel_2 : Channel_830843C1;
	{attribute addProperty Name "Channel_3"}
	Channel_3 : Channel_830843C1;
	{attribute addProperty Name "Channel_4"}
	Channel_4 : Channel_830843C1;
	{attribute addProperty Name "Channel_5"}
	Channel_5 : Channel_830843C1;
	{attribute addProperty Name "Channel_6"}
	Channel_6 : Channel_830843C1;
	{attribute addProperty Name "Channel_7"}
	Channel_7 : Channel_830843C1;
	{attribute addProperty Name "Channel_8"}
	Channel_8 : Channel_830843C1;
	{attribute addProperty Name "Channel_9"}
	Channel_9 : Channel_830843C1;
	{attribute addProperty Name "Channel_10"}
	Channel_10 : Channel_830843C1;
	{attribute addProperty Name "Channel_11"}
	Channel_11 : Channel_830843C1;
	{attribute addProperty Name "Channel_12"}
	Channel_12 : Channel_830843C1;
	{attribute addProperty Name "Channel_13"}
	Channel_13 : Channel_830843C1;
	{attribute addProperty Name "Channel_14"}
	Channel_14 : Channel_830843C1;
	{attribute addProperty Name "Channel_15"}
	Channel_15 : Channel_830843C1;
	{attribute addProperty Name "Channel_16"}
	Channel_16 : Channel_830843C1;
	{attribute addProperty Name "Channel_17"}
	Channel_17 : Channel_42CA91F7;
	{attribute addProperty Name "Channel_18"}
	Channel_18 : Channel_42CA91F7;
	{attribute addProperty Name "Channel_19"}
	Channel_19 : Channel_42CA91F7;
	{attribute addProperty Name "Channel_20"}
	Channel_20 : Channel_42CA91F7;
	{attribute addProperty Name "Channel_21"}
	Channel_21 : Channel_42CA91F7;
	{attribute addProperty Name "Channel_22"}
	Channel_22 : Channel_42CA91F7;
	{attribute addProperty Name "Channel_23"}
	Channel_23 : Channel_42CA91F7;
	{attribute addProperty Name "Channel_24"}
	Channel_24 : Channel_42CA91F7;
	{attribute addProperty Name "Channel_25"}
	Channel_25 : Channel_42CA91F7;
	{attribute addProperty Name "Channel_26"}
	Channel_26 : Channel_42CA91F7;
	{attribute addProperty Name "Channel_27"}
	Channel_27 : Channel_42CA91F7;
	{attribute addProperty Name "Channel_28"}
	Channel_28 : Channel_42CA91F7;
	{attribute addProperty Name "Channel_29"}
	Channel_29 : Channel_42CA91F7;
	{attribute addProperty Name "Channel_30"}
	Channel_30 : Channel_42CA91F7;
	{attribute addProperty Name "Channel_31"}
	Channel_31 : Channel_42CA91F7;
	{attribute addProperty Name "Channel_32"}
	Channel_32 : Channel_42CA91F7;
	{attribute addProperty Name "WcState"}
	WcState : WcState_9091E0EB;
	{attribute addProperty Name "InfoData"}
	InfoData : InfoData_6F19DB2B;
END_STRUCT
END_TYPE

// ---- DUTs/IO/Boxes/ER2624_7B64371E.TcDUT
{attribute 'GeneratedUsingTerminal: ER2624-0002-0018'}
{attribute addProperty BoxType "ER2624-0002-0018"}
{attribute addProperty Description "ER2624-0002 4Ch. Relay Output, NO (125V AC / 30V DC)"}
{attribute addProperty Physics "YY"}
{attribute addProperty Id "Channel_1AT %Q*Channel_42CA91F71Channel_2AT %Q*Channel_42CA91F71Channel_3AT %Q*Channel_42CA91F71Channel_4AT %Q*Channel_42CA91F71WcStateAT %I*WcState_0B2B16F91InfoDataAT %I*InfoData_6F19DB2B2"}
{attribute addProperty CRC "2070165278"}
{attribute addProperty Size "7"}
TYPE ER2624_7B64371E EXTENDS EtcSlaveBoxBase_77A0E4A7 :
STRUCT
	{attribute addProperty Name "Channel_1"}
	Channel_1 : Channel_42CA91F7;
	{attribute addProperty Name "Channel_2"}
	Channel_2 : Channel_42CA91F7;
	{attribute addProperty Name "Channel_3"}
	Channel_3 : Channel_42CA91F7;
	{attribute addProperty Name "Channel_4"}
	Channel_4 : Channel_42CA91F7;
	{attribute addProperty Name "WcState"}
	WcState : WcState_0B2B16F9;
	{attribute addProperty Name "InfoData"}
	InfoData : InfoData_6F19DB2B;
END_STRUCT
END_TYPE

// ---- DUTs/IO/Boxes/ER2809_2B6483BD.TcDUT
{attribute 'GeneratedUsingTerminal: ER2809-0021-0017'}
{attribute addProperty BoxType "ER2809-0021-0017"}
{attribute addProperty Description "ER2809-0021 16 Ch. Dig. Output 24V, 0,5A, M8"}
{attribute addProperty Physics "YY"}
{attribute addProperty Id "Channel_1AT %Q*Channel_42CA91F71Channel_2AT %Q*Channel_42CA91F71Channel_3AT %Q*Channel_42CA91F71Channel_4AT %Q*Channel_42CA91F71Channel_5AT %Q*Channel_42CA91F71Channel_6AT %Q*Channel_42CA91F71Channel_7AT %Q*Channel_42CA91F71Channel_8AT %Q*Channel_42CA91F71Channel_9AT %Q*Channel_42CA91F71Channel_10AT %Q*Channel_42CA91F71Channel_11AT %Q*Channel_42CA91F71Channel_12AT %Q*Channel_42CA91F71Channel_13AT %Q*Channel_42CA91F71Channel_14AT %Q*Channel_42CA91F71Channel_15AT %Q*Channel_42CA91F71Channel_16AT %Q*Channel_42CA91F71WcStateAT %I*WcState_0B2B16F91InfoDataAT %I*InfoData_6F19DB2B2"}
{attribute addProperty CRC "728007613"}
{attribute addProperty Size "19"}
TYPE ER2809_2B6483BD EXTENDS EtcSlaveBoxBase_77A0E4A7 :
STRUCT
	{attribute addProperty Name "Channel_1"}
	Channel_1 : Channel_42CA91F7;
	{attribute addProperty Name "Channel_2"}
	Channel_2 : Channel_42CA91F7;
	{attribute addProperty Name "Channel_3"}
	Channel_3 : Channel_42CA91F7;
	{attribute addProperty Name "Channel_4"}
	Channel_4 : Channel_42CA91F7;
	{attribute addProperty Name "Channel_5"}
	Channel_5 : Channel_42CA91F7;
	{attribute addProperty Name "Channel_6"}
	Channel_6 : Channel_42CA91F7;
	{attribute addProperty Name "Channel_7"}
	Channel_7 : Channel_42CA91F7;
	{attribute addProperty Name "Channel_8"}
	Channel_8 : Channel_42CA91F7;
	{attribute addProperty Name "Channel_9"}
	Channel_9 : Channel_42CA91F7;
	{attribute addProperty Name "Channel_10"}
	Channel_10 : Channel_42CA91F7;
	{attribute addProperty Name "Channel_11"}
	Channel_11 : Channel_42CA91F7;
	{attribute addProperty Name "Channel_12"}
	Channel_12 : Channel_42CA91F7;
	{attribute addProperty Name "Channel_13"}
	Channel_13 : Channel_42CA91F7;
	{attribute addProperty Name "Channel_14"}
	Channel_14 : Channel_42CA91F7;
	{attribute addProperty Name "Channel_15"}
	Channel_15 : Channel_42CA91F7;
	{attribute addProperty Name "Channel_16"}
	Channel_16 : Channel_42CA91F7;
	{attribute addProperty Name "WcState"}
	WcState : WcState_0B2B16F9;
	{attribute addProperty Name "InfoData"}
	InfoData : InfoData_6F19DB2B;
END_STRUCT
END_TYPE

// ---- DUTs/IO/Boxes/ER3174_DCC78662.TcDUT
{attribute 'GeneratedUsingTerminal: ER3174-0002-0016'}
{attribute addProperty BoxType "ER3174-0002-0016"}
{attribute addProperty Description "ER3174-0002 4Ch. Ana. Input +/-10V, 0-10V, 0/4-20mA configurable"}
{attribute addProperty Physics "YY"}
{attribute addProperty Id "AI_Standard_Channel_1AT %I*AI_Standard_Channel_A8DF64E310AI_Standard_Channel_2AT %I*AI_Standard_Channel_A8DF64E310AI_Standard_Channel_3AT %I*AI_Standard_Channel_A8DF64E310AI_Standard_Channel_4AT %I*AI_Standard_Channel_A8DF64E310WcStateAT %I*WcState_9091E0EB2InfoDataAT %I*InfoData_32EB74EA10"}
{attribute addProperty CRC "3704063586"}
{attribute addProperty Size "52"}
TYPE ER3174_DCC78662 EXTENDS EtcSlaveBoxBase_77A0E4A7 :
STRUCT
	{attribute addProperty Name "AI_Standard_Channel_1"}
	AI_Standard_Channel_1 : AI_Standard_Channel_A8DF64E3;
	{attribute addProperty Name "AI_Standard_Channel_2"}
	AI_Standard_Channel_2 : AI_Standard_Channel_A8DF64E3;
	{attribute addProperty Name "AI_Standard_Channel_3"}
	AI_Standard_Channel_3 : AI_Standard_Channel_A8DF64E3;
	{attribute addProperty Name "AI_Standard_Channel_4"}
	AI_Standard_Channel_4 : AI_Standard_Channel_A8DF64E3;
	{attribute addProperty Name "WcState"}
	WcState : WcState_9091E0EB;
	{attribute addProperty Name "InfoData"}
	InfoData : InfoData_32EB74EA;
END_STRUCT
END_TYPE

// ---- DUTs/IO/Boxes/ER3184_DCC78662.TcDUT
{attribute 'GeneratedUsingTerminal: ER3184-0002-0019'}
{attribute addProperty BoxType "ER3184-0002-0019"}
{attribute addProperty Description "ER3184-0002 4Ch. Ana. Input +/-10V, 0-10V, 0/4-20mA configurable, single ended"}
{attribute addProperty Physics "YY"}
{attribute addProperty Id "AI_Standard_Channel_1AT %I*AI_Standard_Channel_A8DF64E310AI_Standard_Channel_2AT %I*AI_Standard_Channel_A8DF64E310AI_Standard_Channel_3AT %I*AI_Standard_Channel_A8DF64E310AI_Standard_Channel_4AT %I*AI_Standard_Channel_A8DF64E310WcStateAT %I*WcState_9091E0EB2InfoDataAT %I*InfoData_32EB74EA10"}
{attribute addProperty CRC "3704063586"}
{attribute addProperty Size "52"}
TYPE ER3184_DCC78662 EXTENDS EtcSlaveBoxBase_77A0E4A7 :
STRUCT
	{attribute addProperty Name "AI_Standard_Channel_1"}
	AI_Standard_Channel_1 : AI_Standard_Channel_A8DF64E3;
	{attribute addProperty Name "AI_Standard_Channel_2"}
	AI_Standard_Channel_2 : AI_Standard_Channel_A8DF64E3;
	{attribute addProperty Name "AI_Standard_Channel_3"}
	AI_Standard_Channel_3 : AI_Standard_Channel_A8DF64E3;
	{attribute addProperty Name "AI_Standard_Channel_4"}
	AI_Standard_Channel_4 : AI_Standard_Channel_A8DF64E3;
	{attribute addProperty Name "WcState"}
	WcState : WcState_9091E0EB;
	{attribute addProperty Name "InfoData"}
	InfoData : InfoData_32EB74EA;
END_STRUCT
END_TYPE

// ---- DUTs/IO/Boxes/ER3204_6CD7E119.TcDUT
{attribute 'GeneratedUsingTerminal: ER3204-0002-0016'}
{attribute addProperty BoxType "ER3204-0002-0016"}
{attribute addProperty Description "ER3204-0002 4Ch. Ana. Input PT100 (RTD)"}
{attribute addProperty Physics "YY"}
{attribute addProperty Id "RTD_RTDInputs_Channel_1AT %I*RTD_RTDInputs_Channel_A8DF64E310RTD_RTDInputs_Channel_2AT %I*RTD_RTDInputs_Channel_A8DF64E310RTD_RTDInputs_Channel_3AT %I*RTD_RTDInputs_Channel_A8DF64E310RTD_RTDInputs_Channel_4AT %I*RTD_RTDInputs_Channel_A8DF64E310WcStateAT %I*WcState_9091E0EB2InfoDataAT %I*InfoData_32EB74EA10"}
{attribute addProperty CRC "1826087193"}
{attribute addProperty Size "52"}
TYPE ER3204_6CD7E119 EXTENDS EtcSlaveBoxBase_77A0E4A7 :
STRUCT
	{attribute addProperty Name "RTD_RTDInputs_Channel_1"}
	RTD_RTDInputs_Channel_1 : RTD_RTDInputs_Channel_A8DF64E3;
	{attribute addProperty Name "RTD_RTDInputs_Channel_2"}
	RTD_RTDInputs_Channel_2 : RTD_RTDInputs_Channel_A8DF64E3;
	{attribute addProperty Name "RTD_RTDInputs_Channel_3"}
	RTD_RTDInputs_Channel_3 : RTD_RTDInputs_Channel_A8DF64E3;
	{attribute addProperty Name "RTD_RTDInputs_Channel_4"}
	RTD_RTDInputs_Channel_4 : RTD_RTDInputs_Channel_A8DF64E3;
	{attribute addProperty Name "WcState"}
	WcState : WcState_9091E0EB;
	{attribute addProperty Name "InfoData"}
	InfoData : InfoData_32EB74EA;
END_STRUCT
END_TYPE

// ---- DUTs/IO/Boxes/ER3204_AB25C3AC.TcDUT
{attribute 'GeneratedUsingTerminal: ER3204-0002-0021'}
{attribute addProperty BoxType "ER3204-0002-0021"}
{attribute addProperty Description "ER3204-0002 4Ch. Ana. Input PT100 (RTD)"}
{attribute addProperty Physics "YY"}
{attribute addProperty Id "RTD_RTDInputs_Channel_1AT %I*AI_Standard_Channel_4A3944819RTD_RTDInputs_Channel_2AT %I*AI_Standard_Channel_4A3944819RTD_RTDInputs_Channel_3AT %I*AI_Standard_Channel_4A3944819RTD_RTDInputs_Channel_4AT %I*AI_Standard_Channel_4A3944819WcStateAT %I*WcState_9091E0EB2InfoDataAT %I*InfoData_32EB74EA10"}
{attribute addProperty CRC "2871378860"}
{attribute addProperty Size "48"}
TYPE ER3204_AB25C3AC EXTENDS EtcSlaveBoxBase_77A0E4A7 :
STRUCT
	{attribute addProperty Name "RTD_RTDInputs_Channel_1"}
	RTD_RTDInputs_Channel_1 : AI_Standard_Channel_4A394481;
	{attribute addProperty Name "RTD_RTDInputs_Channel_2"}
	RTD_RTDInputs_Channel_2 : AI_Standard_Channel_4A394481;
	{attribute addProperty Name "RTD_RTDInputs_Channel_3"}
	RTD_RTDInputs_Channel_3 : AI_Standard_Channel_4A394481;
	{attribute addProperty Name "RTD_RTDInputs_Channel_4"}
	RTD_RTDInputs_Channel_4 : AI_Standard_Channel_4A394481;
	{attribute addProperty Name "WcState"}
	WcState : WcState_9091E0EB;
	{attribute addProperty Name "InfoData"}
	InfoData : InfoData_32EB74EA;
END_STRUCT
END_TYPE

// ---- DUTs/IO/Boxes/ER3314_E65CDB1C.TcDUT
{attribute 'GeneratedUsingTerminal: ER3314-0002-0021'}
{attribute addProperty BoxType "ER3314-0002-0021"}
{attribute addProperty Description "ER3314-0002 4Ch. Ana. Input Thermocouple (TC)"}
{attribute addProperty Physics "YY"}
{attribute addProperty Id "TC_Inputs_Channel_1AT %I*AI_Standard_Channel_4A3944819TC_Inputs_Channel_2AT %I*AI_Standard_Channel_4A3944819TC_Inputs_Channel_3AT %I*AI_Standard_Channel_4A3944819TC_Inputs_Channel_4AT %I*AI_Standard_Channel_4A3944819WcStateAT %I*WcState_9091E0EB2InfoDataAT %I*InfoData_32EB74EA10"}
{attribute addProperty CRC "3864845084"}
{attribute addProperty Size "48"}
TYPE ER3314_E65CDB1C EXTENDS EtcSlaveBoxBase_77A0E4A7 :
STRUCT
	{attribute addProperty Name "TC_Inputs_Channel_1"}
	TC_Inputs_Channel_1 : AI_Standard_Channel_4A394481;
	{attribute addProperty Name "TC_Inputs_Channel_2"}
	TC_Inputs_Channel_2 : AI_Standard_Channel_4A394481;
	{attribute addProperty Name "TC_Inputs_Channel_3"}
	TC_Inputs_Channel_3 : AI_Standard_Channel_4A394481;
	{attribute addProperty Name "TC_Inputs_Channel_4"}
	TC_Inputs_Channel_4 : AI_Standard_Channel_4A394481;
	{attribute addProperty Name "WcState"}
	WcState : WcState_9091E0EB;
	{attribute addProperty Name "InfoData"}
	InfoData : InfoData_32EB74EA;
END_STRUCT
END_TYPE

// ---- DUTs/IO/Boxes/ER4174_AB92710E.TcDUT
{attribute 'GeneratedUsingTerminal: ER4174-0002-0016'}
{attribute addProperty BoxType "ER4174-0002-0016"}
{attribute addProperty Description "ER4174-0002 4Ch. Ana. Output +/-10V, 0-10V, 0/4-20mA configurable"}
{attribute addProperty Physics "YY"}
{attribute addProperty Id "AO_Outputs_Channel_1AT %Q*AO_Output_Channel_BA7EBB7C2AO_Outputs_Channel_2AT %Q*AO_Output_Channel_BA7EBB7C2AO_Outputs_Channel_3AT %Q*AO_Output_Channel_BA7EBB7C2AO_Outputs_Channel_4AT %Q*AO_Output_Channel_BA7EBB7C2WcStateAT %I*WcState_0B2B16F91InfoDataAT %I*InfoData_32EB74EA10"}
{attribute addProperty CRC "2878501134"}
{attribute addProperty Size "19"}
TYPE ER4174_AB92710E EXTENDS EtcSlaveBoxBase_77A0E4A7 :
STRUCT
	{attribute addProperty Name "AO_Outputs_Channel_1"}
	AO_Outputs_Channel_1 : AO_Output_Channel_BA7EBB7C;
	{attribute addProperty Name "AO_Outputs_Channel_2"}
	AO_Outputs_Channel_2 : AO_Output_Channel_BA7EBB7C;
	{attribute addProperty Name "AO_Outputs_Channel_3"}
	AO_Outputs_Channel_3 : AO_Output_Channel_BA7EBB7C;
	{attribute addProperty Name "AO_Outputs_Channel_4"}
	AO_Outputs_Channel_4 : AO_Output_Channel_BA7EBB7C;
	{attribute addProperty Name "WcState"}
	WcState : WcState_0B2B16F9;
	{attribute addProperty Name "InfoData"}
	InfoData : InfoData_32EB74EA;
END_STRUCT
END_TYPE

// ---- DUTs/IO/Boxes/ER4374_A304750F.TcDUT
{attribute 'GeneratedUsingTerminal: ER4374-0002-0018'}
{attribute addProperty BoxType "ER4374-0002-0018"}
{attribute addProperty Description "ER4374-0002 2Ch. Ana. Input +/-10V, 0-10V, 0/4-20mA configurable; 2Ch. Ana. Output +/-10V, 0-10V, 0/4-20mA configurable"}
{attribute addProperty Physics "YY"}
{attribute addProperty Id "AI_Inputs_Channel_1AT %I*AI_Inputs_Channel_A8DF64E310AI_Inputs_Channel_2AT %I*AI_Inputs_Channel_A8DF64E310AO_Outputs_Channel_3AT %Q*AO_Output_Channel_BA7EBB7C2AO_Outputs_Channel_4AT %Q*AO_Output_Channel_BA7EBB7C2WcStateAT %I*WcState_9091E0EB2InfoDataAT %I*InfoData_32EB74EA10"}
{attribute addProperty CRC "2734978319"}
{attribute addProperty Size "36"}
TYPE ER4374_A304750F EXTENDS EtcSlaveBoxBase_77A0E4A7 :
STRUCT
	{attribute addProperty Name "AI_Inputs_Channel_1"}
	AI_Inputs_Channel_1 : AI_Inputs_Channel_A8DF64E3;
	{attribute addProperty Name "AI_Inputs_Channel_2"}
	AI_Inputs_Channel_2 : AI_Inputs_Channel_A8DF64E3;
	{attribute addProperty Name "AO_Outputs_Channel_3"}
	AO_Outputs_Channel_3 : AO_Output_Channel_BA7EBB7C;
	{attribute addProperty Name "AO_Outputs_Channel_4"}
	AO_Outputs_Channel_4 : AO_Output_Channel_BA7EBB7C;
	{attribute addProperty Name "WcState"}
	WcState : WcState_9091E0EB;
	{attribute addProperty Name "InfoData"}
	InfoData : InfoData_32EB74EA;
END_STRUCT
END_TYPE

// ---- DUTs/IO/Boxes/ER5101_87AC78CF.TcDUT
{attribute 'GeneratedUsingTerminal: ER5101-0002-0019'}
{attribute addProperty BoxType "ER5101-0002-0019"}
{attribute addProperty Description "ER5101-0002 1Ch. Inc. Encoder 5V, M12"}
{attribute addProperty Physics "YY"}
{attribute addProperty Id "ENC_Status_compactAT %I*ENC_Status_compact_F4F8958316ENC_Control_compactAT %Q*ENC_Control_compact_E6DC9B254WcStateAT %I*WcState_9091E0EB2InfoDataAT %I*InfoData_32EB74EA10"}
{attribute addProperty CRC "2276227279"}
{attribute addProperty Size "32"}
TYPE ER5101_87AC78CF EXTENDS EtcSlaveBoxBase_77A0E4A7 :
STRUCT
	{attribute addProperty Name "ENC_Status_compact"}
	ENC_Status_compact : ENC_Status_compact_F4F89583;
	{attribute addProperty Name "ENC_Control_compact"}
	ENC_Control_compact : ENC_Control_compact_E6DC9B25;
	{attribute addProperty Name "WcState"}
	WcState : WcState_9091E0EB;
	{attribute addProperty Name "InfoData"}
	InfoData : InfoData_32EB74EA;
END_STRUCT
END_TYPE

// ---- DUTs/IO/Boxes/ER5151_7476E948.TcDUT
{attribute 'GeneratedUsingTerminal: ER5151-0002-0018'}
{attribute addProperty BoxType "ER5151-0002-0018"}
{attribute addProperty Description "ER5151-0002 1Ch. Inc. Encoder 24V, M12, single ended"}
{attribute addProperty Physics "YY"}
{attribute addProperty Id "ENC_Status_compactAT %I*ENC_Status_compact_7D3464F320ENC_Control_compactAT %Q*ENC_Control_compact_21E2D14D6WcStateAT %I*WcState_9091E0EB2InfoDataAT %I*InfoData_32EB74EA10"}
{attribute addProperty CRC "1953950024"}
{attribute addProperty Size "38"}
TYPE ER5151_7476E948 EXTENDS EtcSlaveBoxBase_77A0E4A7 :
STRUCT
	{attribute addProperty Name "ENC_Status_compact"}
	ENC_Status_compact : ENC_Status_compact_7D3464F3;
	{attribute addProperty Name "ENC_Control_compact"}
	ENC_Control_compact : ENC_Control_compact_21E2D14D;
	{attribute addProperty Name "WcState"}
	WcState : WcState_9091E0EB;
	{attribute addProperty Name "InfoData"}
	InfoData : InfoData_32EB74EA;
END_STRUCT
END_TYPE

// ---- DUTs/IO/Boxes/ER6001_40883D03.TcDUT
{attribute 'GeneratedUsingTerminal: ER6001-0002-0016'}
{attribute addProperty BoxType "ER6001-0002-0016"}
{attribute addProperty Description "ER6001-0002 Interface (RS232/422/485)"}
{attribute addProperty Physics "YY"}
{attribute addProperty Id "COM_InputsAT %I*COM_Inputs_6C2FC20224COM_OutputsAT %Q*COM_Outputs_5D00B5E724WcStateAT %I*WcState_9091E0EB2InfoDataAT %I*InfoData_32EB74EA10"}
{attribute addProperty CRC "1082670339"}
{attribute addProperty Size "60"}
TYPE ER6001_40883D03 EXTENDS EtcSlaveBoxBase_77A0E4A7 :
STRUCT
	{attribute addProperty Name "COM_Inputs"}
	COM_Inputs : COM_Inputs_6C2FC202;
	{attribute addProperty Name "COM_Outputs"}
	COM_Outputs : COM_Outputs_5D00B5E7;
	{attribute addProperty Name "WcState"}
	WcState : WcState_9091E0EB;
	{attribute addProperty Name "InfoData"}
	InfoData : InfoData_32EB74EA;
END_STRUCT
END_TYPE

// ---- DUTs/IO/Boxes/ER6002_7F53816A.TcDUT
{attribute 'GeneratedUsingTerminal: ER6002-0002-0021'}
{attribute addProperty BoxType "ER6002-0002-0021"}
{attribute addProperty Description "ER6002-0002 Interface (RS232/422/485)"}
{attribute addProperty Physics "YY"}
{attribute addProperty Id "COM_TxPDO_Map_Inputs_Channel_1AT %I*COM_TxPDO_Map_Inputs_Channel_C252EAC224COM_TxPDO_Map_Inputs_Channel_2AT %I*COM_TxPDO_Map_Inputs_Channel_C252EAC224COM_RxPDO_Map_Outputs_Channel_1AT %Q*COM_RxPDO_Map_Outputs_Channel_B336F4EE24COM_RxPDO_Map_Outputs_Channel_2AT %Q*COM_RxPDO_Map_Outputs_Channel_B336F4EE24WcStateAT %I*WcState_9091E0EB2InfoDataAT %I*InfoData_32EB74EA10"}
{attribute addProperty CRC "2136179050"}
{attribute addProperty Size "108"}
TYPE ER6002_7F53816A EXTENDS EtcSlaveBoxBase_77A0E4A7 :
STRUCT
	{attribute addProperty Name "COM_TxPDO_Map_Inputs_Channel_1"}
	COM_TxPDO_Map_Inputs_Channel_1 : COM_TxPDO_Map_Inputs_Channel_C252EAC2;
	{attribute addProperty Name "COM_TxPDO_Map_Inputs_Channel_2"}
	COM_TxPDO_Map_Inputs_Channel_2 : COM_TxPDO_Map_Inputs_Channel_C252EAC2;
	{attribute addProperty Name "COM_RxPDO_Map_Outputs_Channel_1"}
	COM_RxPDO_Map_Outputs_Channel_1 : COM_RxPDO_Map_Outputs_Channel_B336F4EE;
	{attribute addProperty Name "COM_RxPDO_Map_Outputs_Channel_2"}
	COM_RxPDO_Map_Outputs_Channel_2 : COM_RxPDO_Map_Outputs_Channel_B336F4EE;
	{attribute addProperty Name "WcState"}
	WcState : WcState_9091E0EB;
	{attribute addProperty Name "InfoData"}
	InfoData : InfoData_32EB74EA;
END_STRUCT
END_TYPE

// ---- DUTs/IO/Boxes/ER6002_7BE6B617.TcDUT
{attribute 'GeneratedUsingTerminal: ER6002-0002-0022'}
{attribute addProperty BoxType "ER6002-0002-0022"}
{attribute addProperty Description "ER6002-0002 Interface (RS232/422/485)"}
{attribute addProperty Physics "YY"}
{attribute addProperty Id "COM_TxPDO_Map_Inputs_Channel_1AT %I*COM_TxPDO_Map_Inputs_Channel_6C2FC20224COM_TxPDO_Map_Inputs_Channel_2AT %I*COM_TxPDO_Map_Inputs_Channel_6C2FC20224COM_RxPDO_Map_Outputs_Channel_1AT %Q*COM_RxPDO_Map_Outputs_Channel_5D00B5E724COM_RxPDO_Map_Outputs_Channel_2AT %Q*COM_RxPDO_Map_Outputs_Channel_5D00B5E724WcStateAT %I*WcState_9091E0EB2InfoDataAT %I*InfoData_32EB74EA10"}
{attribute addProperty CRC "2078717463"}
{attribute addProperty Size "108"}
TYPE ER6002_7BE6B617 EXTENDS EtcSlaveBoxBase_77A0E4A7 :
STRUCT
	{attribute addProperty Name "COM_TxPDO_Map_Inputs_Channel_1"}
	COM_TxPDO_Map_Inputs_Channel_1 : COM_TxPDO_Map_Inputs_Channel_6C2FC202;
	{attribute addProperty Name "COM_TxPDO_Map_Inputs_Channel_2"}
	COM_TxPDO_Map_Inputs_Channel_2 : COM_TxPDO_Map_Inputs_Channel_6C2FC202;
	{attribute addProperty Name "COM_RxPDO_Map_Outputs_Channel_1"}
	COM_RxPDO_Map_Outputs_Channel_1 : COM_RxPDO_Map_Outputs_Channel_5D00B5E7;
	{attribute addProperty Name "COM_RxPDO_Map_Outputs_Channel_2"}
	COM_RxPDO_Map_Outputs_Channel_2 : COM_RxPDO_Map_Outputs_Channel_5D00B5E7;
	{attribute addProperty Name "WcState"}
	WcState : WcState_9091E0EB;
	{attribute addProperty Name "InfoData"}
	InfoData : InfoData_32EB74EA;
END_STRUCT
END_TYPE

// ---- DUTs/IO/Boxes/ER7041_3210CF40.TcDUT
{attribute 'GeneratedUsingTerminal: ER7041-0002-0024'}
{attribute addProperty BoxType "ER7041-0002-0024"}
{attribute addProperty Description "ER7041-0002 1Ch. Stepper motor output stage (50V, 5A)"}
{attribute addProperty Physics "YY"}
{attribute addProperty Id "ENC_Status_compactAT %I*ENC_Status_compact_4D066E1A16STM_StatusAT %I*STM_Status_36ED096F11ENC_Control_compactAT %Q*ENC_Control_compact_21E2D14D6STM_ControlAT %Q*STM_Control_BA4CE3524STM_VelocityAT %Q*STM_Velocity_A47A3F412WcStateAT %I*WcState_9091E0EB2InfoDataAT %I*InfoData_6538CF5F12"}
{attribute addProperty CRC "839962432"}
{attribute addProperty Size "53"}
TYPE ER7041_3210CF40 EXTENDS EtcSlaveBoxBase_77A0E4A7 :
STRUCT
	{attribute addProperty Name "ENC_Status_compact"}
	ENC_Status_compact : ENC_Status_compact_4D066E1A;
	{attribute addProperty Name "STM_Status"}
	STM_Status : STM_Status_36ED096F;
	{attribute addProperty Name "ENC_Control_compact"}
	ENC_Control_compact : ENC_Control_compact_21E2D14D;
	{attribute addProperty Name "STM_Control"}
	STM_Control : STM_Control_BA4CE352;
	{attribute addProperty Name "STM_Velocity"}
	STM_Velocity : STM_Velocity_A47A3F41;
	{attribute addProperty Name "WcState"}
	WcState : WcState_9091E0EB;
	{attribute addProperty Name "InfoData"}
	InfoData : InfoData_6538CF5F;
END_STRUCT
END_TYPE

// ---- DUTs/IO/Boxes/ER7041_3E4BEAEF.TcDUT
{attribute 'GeneratedUsingTerminal: ER7041-3002-0021'}
{attribute addProperty BoxType "ER7041-3002-0021"}
{attribute addProperty Description "ER7041-3002 1Ch. Stepper motor output stage (50V, 5A)"}
{attribute addProperty Physics "YY"}
{attribute addProperty Id "ENC_Status_compactAT %I*ENC_Status_compact_4D066E1A16STM_StatusAT %I*STM_Status_DE0D6B3712ENC_Control_compactAT %Q*ENC_Control_compact_21E2D14D6STM_ControlAT %Q*STM_Control_BA4CE3524STM_VelocityAT %Q*STM_Velocity_A47A3F412WcStateAT %I*WcState_9091E0EB2InfoDataAT %I*InfoData_6538CF5F12"}
{attribute addProperty CRC "1045162735"}
{attribute addProperty Size "54"}
TYPE ER7041_3E4BEAEF EXTENDS EtcSlaveBoxBase_77A0E4A7 :
STRUCT
	{attribute addProperty Name "ENC_Status_compact"}
	ENC_Status_compact : ENC_Status_compact_4D066E1A;
	{attribute addProperty Name "STM_Status"}
	STM_Status : STM_Status_DE0D6B37;
	{attribute addProperty Name "ENC_Control_compact"}
	ENC_Control_compact : ENC_Control_compact_21E2D14D;
	{attribute addProperty Name "STM_Control"}
	STM_Control : STM_Control_BA4CE352;
	{attribute addProperty Name "STM_Velocity"}
	STM_Velocity : STM_Velocity_A47A3F41;
	{attribute addProperty Name "WcState"}
	WcState : WcState_9091E0EB;
	{attribute addProperty Name "InfoData"}
	InfoData : InfoData_6538CF5F;
END_STRUCT
END_TYPE

// ---- DUTs/IO/Boxes/ER7342_2AE9C6B3.TcDUT
{attribute 'GeneratedUsingTerminal: ER7342-0002-0020'}
{attribute addProperty BoxType "ER7342-0002-0020"}
{attribute addProperty Description "ER7342-0002 2Ch. DC motor output stage (50V, 3.5A)"}
{attribute addProperty Physics "YY"}
{attribute addProperty Id "ENC_Status_compact_Channel_1AT %I*ENC_Status_compact_Channel_DC559AB014ENC_Status_compact_Channel_2AT %I*ENC_Status_compact_Channel_DC559AB014DCM_Status_Channel_1AT %I*DCM_Status_Channel_36ED096F11DCM_Status_Channel_2AT %I*DCM_Status_Channel_36ED096F11ENC_Control_compact_Channel_1AT %Q*ENC_Control_compact_Channel_2E82BC435ENC_Control_compact_Channel_2AT %Q*ENC_Control_compact_Channel_2E82BC435DCM_Control_Channel_1AT %Q*DCM_Control_Channel_5A8B50163DCM_Velocity_Channel_1AT %Q*DCM_Velocity_Channel_A47A3F412DCM_Control_Channel_2AT %Q*DCM_Control_Channel_5A8B50163DCM_Velocity_Channel_2AT %Q*DCM_Velocity_Channel_A47A3F412WcStateAT %I*WcState_9091E0EB2InfoDataAT %I*InfoData_939F71B614"}
{attribute addProperty CRC "719963827"}
{attribute addProperty Size "86"}
TYPE ER7342_2AE9C6B3 EXTENDS EtcSlaveBoxBase_77A0E4A7 :
STRUCT
	{attribute addProperty Name "ENC_Status_compact_Channel_1"}
	ENC_Status_compact_Channel_1 : ENC_Status_compact_Channel_DC559AB0;
	{attribute addProperty Name "ENC_Status_compact_Channel_2"}
	ENC_Status_compact_Channel_2 : ENC_Status_compact_Channel_DC559AB0;
	{attribute addProperty Name "DCM_Status_Channel_1"}
	DCM_Status_Channel_1 : DCM_Status_Channel_36ED096F;
	{attribute addProperty Name "DCM_Status_Channel_2"}
	DCM_Status_Channel_2 : DCM_Status_Channel_36ED096F;
	{attribute addProperty Name "ENC_Control_compact_Channel_1"}
	ENC_Control_compact_Channel_1 : ENC_Control_compact_Channel_2E82BC43;
	{attribute addProperty Name "ENC_Control_compact_Channel_2"}
	ENC_Control_compact_Channel_2 : ENC_Control_compact_Channel_2E82BC43;
	{attribute addProperty Name "DCM_Control_Channel_1"}
	DCM_Control_Channel_1 : DCM_Control_Channel_5A8B5016;
	{attribute addProperty Name "DCM_Velocity_Channel_1"}
	DCM_Velocity_Channel_1 : DCM_Velocity_Channel_A47A3F41;
	{attribute addProperty Name "DCM_Control_Channel_2"}
	DCM_Control_Channel_2 : DCM_Control_Channel_5A8B5016;
	{attribute addProperty Name "DCM_Velocity_Channel_2"}
	DCM_Velocity_Channel_2 : DCM_Velocity_Channel_A47A3F41;
	{attribute addProperty Name "WcState"}
	WcState : WcState_9091E0EB;
	{attribute addProperty Name "InfoData"}
	InfoData : InfoData_939F71B6;
END_STRUCT
END_TYPE

// ---- DUTs/IO/Boxes/ER8309_A0C54F77.TcDUT
{attribute 'GeneratedUsingTerminal: ER8309-1022-0018'}
{attribute addProperty BoxType "ER8309-1022-0018"}
{attribute addProperty Description "ER8309-1022 2Ch. Ana. Input 4-20mA, 1Ch. Pulse Width Current Output (24V, 1.2A), 1 Ch Ana. Output, 2Ch Dig. Out 24V, 0.5A, 4Ch Dig. In. 24V, 4Ch Dig In/Out 24V, 0.5A, M12"}
{attribute addProperty Physics "YY"}
{attribute addProperty Id "AI_Inputs_Channel_1AT %I*AI_Inputs_Channel_A8DF64E310AI_Inputs_Channel_2AT %I*AI_Inputs_Channel_A8DF64E310TACHO_Single_Shaft_Mode_Input_Channel_1AT %I*TACHO_Single_Shaft_Mode_Input_Channel_C331CA3E10DIG_InputsAT %I*DIG_Inputs_495F5DA48PWM_StatusAT %I*PWM_Status_77939B114DEV_InputsAT %I*DEV_Inputs_FBF180A42TACHO_Output_Channel_1AT %Q*TACHO_Output_Channel_600697D91DIG_OutputsAT %Q*DIG_Outputs_0E2843948PWM_ControlAT %Q*PWM_Control_63F162E45WcStateAT %I*WcState_9091E0EB2InfoDataAT %I*InfoData_32EB74EA10"}
{attribute addProperty CRC "2697285495"}
{attribute addProperty Size "70"}
TYPE ER8309_A0C54F77 EXTENDS EtcSlaveBoxBase_77A0E4A7 :
STRUCT
	{attribute addProperty Name "AI_Inputs_Channel_1"}
	AI_Inputs_Channel_1 : AI_Inputs_Channel_A8DF64E3;
	{attribute addProperty Name "AI_Inputs_Channel_2"}
	AI_Inputs_Channel_2 : AI_Inputs_Channel_A8DF64E3;
	{attribute addProperty Name "TACHO_Single_Shaft_Mode_Input_Channel_1"}
	TACHO_Single_Shaft_Mode_Input_Channel_1 : TACHO_Single_Shaft_Mode_Input_Channel_C331CA3E;
	{attribute addProperty Name "DIG_Inputs"}
	DIG_Inputs : DIG_Inputs_495F5DA4;
	{attribute addProperty Name "PWM_Status"}
	PWM_Status : PWM_Status_77939B11;
	{attribute addProperty Name "DEV_Inputs"}
	DEV_Inputs : DEV_Inputs_FBF180A4;
	{attribute addProperty Name "TACHO_Output_Channel_1"}
	TACHO_Output_Channel_1 : TACHO_Output_Channel_600697D9;
	{attribute addProperty Name "DIG_Outputs"}
	DIG_Outputs : DIG_Outputs_0E284394;
	{attribute addProperty Name "PWM_Control"}
	PWM_Control : PWM_Control_63F162E4;
	{attribute addProperty Name "WcState"}
	WcState : WcState_9091E0EB;
	{attribute addProperty Name "InfoData"}
	InfoData : InfoData_32EB74EA;
END_STRUCT
END_TYPE

// ---- DUTs/IO/Devices/SyncUnitTask_2D604ED5.TcDUT
{attribute 'GeneratedUsingTerminal: IODEVICETYPE_ETHERCATPROT'}
{attribute addProperty BoxType "IODEVICETYPE_ETHERCATPROT"}
{attribute addProperty Id "WcStateAT %I*WcState_0B2B16F91InfoDataAT %I*InfoData_2A97D6CF8"}
{attribute addProperty CRC "761286357"}
{attribute addProperty Size "9"}
TYPE SyncUnitTask_2D604ED5 :
STRUCT
	{attribute addProperty Name "WcState"}
	WcState : WcState_0B2B16F9;
	{attribute addProperty Name "InfoData"}
	InfoData : InfoData_2A97D6CF;
END_STRUCT
END_TYPE

// ---- DUTs/IO/Devices/SyncUnitTasks_6FEB8257.TcDUT
{attribute 'GeneratedUsingTerminal: '}
{attribute addProperty BoxType ""}
{attribute addProperty Id "unreferencedAT %I*SyncUnitTask_2D604ED59PlcTaskAT %I*SyncUnitTask_2D604ED59"}
{attribute addProperty CRC "1877705303"}
{attribute addProperty Size "18"}
TYPE SyncUnitTasks_6FEB8257 :
STRUCT
	{attribute addProperty Name "unreferenced"}
	unreferenced : SyncUnitTask_2D604ED5;
	{attribute addProperty Name "PlcTask"}
	PlcTask : SyncUnitTask_2D604ED5;
END_STRUCT
END_TYPE

// ---- DUTs/IO/Devices/SyncUnits_99E584AF.TcDUT
{attribute 'GeneratedUsingTerminal: '}
{attribute addProperty BoxType ""}
{attribute addProperty Id "_defaultAT %I*SyncUnitTasks_6FEB825718"}
{attribute addProperty CRC "2581955759"}
{attribute addProperty Size "18"}
TYPE SyncUnits_99E584AF :
STRUCT
	{attribute addProperty Name "_default"}
	_default : SyncUnitTasks_6FEB8257;
END_STRUCT
END_TYPE

// ---- DUTs/IO/Topology/Beckhoff_ER1xxxEK1122_4914C526.TcDUT
{attribute 'GeneratedUsingTerminal: EK1122-0000-0018'}
{attribute addProperty BoxType "EK1122-0000-0018"}
{attribute addProperty Id "Beckhoff_ER1xxxsub_EK1100EK1100_1FC0878B2A_0001_ER1008_0001_0016ER1008_78E8D3DD12A_0002_ER1008_0001_0018ER1008_78E8D3DD12A_0003_ER1008_0002_0018ER1008_78E8D3DD12A_0004_ER1008_0022_0017ER1008_78E8D3DD12A_0005_ER1018_0001_0018ER1018_78E8D3DD12A_0006_ER1018_0002_0018ER1018_78E8D3DD12A_0007_ER1098_0001_0017ER1098_78E8D3DD12A_0008_ER1258_0001_0019ER1258_58F475DD56A_0009_ER1258_0001_0020ER1258_58F475DD56A_0010_ER1258_0002_0019ER1258_58F475DD56A_0011_ER1258_0002_0020ER1258_58F475DD56A_0012_ER1518_0002_0018ER1518_CC44258859A_0013_ER1518_0002_0019ER1518_CC44258859A_0014_ER1809_0021_0017ER1809_32157CFD20A_0015_ER1809_0022_0018ER1809_32157CFD20A_0016_ER1819_0021_0017ER1819_32157CFD20A_0017_ER1819_0022_0017ER1819_32157CFD20"}
{attribute addProperty CRC "1226097958"}
{attribute addProperty Size "508"}
{attribute addProperty Name "Beckhoff ER1xxxEK1122"}
TYPE Beckhoff_ER1xxxEK1122_4914C526 EXTENDS EK1122_1FC0878B :
STRUCT
	{attribute addProperty Name "Beckhoff ER1xxxsub EK1100"}
	{attribute addProperty PreviousPort "Beckhoff ER1xxxEK1122 : D"}
	Beckhoff_ER1xxxsub_EK1100 : EK1100_1FC0878B;
	{attribute addProperty Name "A_0001(ER1008-0001-0016)"}
	{attribute addProperty PreviousPort "Beckhoff ER1xxxsub EK1100 : C"}
	A_0001_ER1008_0001_0016 : ER1008_78E8D3DD;
	{attribute addProperty Name "A_0002(ER1008-0001-0018)"}
	{attribute addProperty PreviousPort "A_0001(ER1008-0001-0016) : B"}
	A_0002_ER1008_0001_0018 : ER1008_78E8D3DD;
	{attribute addProperty Name "A_0003(ER1008-0002-0018)"}
	{attribute addProperty PreviousPort "A_0002(ER1008-0001-0018) : B"}
	A_0003_ER1008_0002_0018 : ER1008_78E8D3DD;
	{attribute addProperty Name "A_0004(ER1008-0022-0017)"}
	{attribute addProperty PreviousPort "A_0003(ER1008-0002-0018) : B"}
	A_0004_ER1008_0022_0017 : ER1008_78E8D3DD;
	{attribute addProperty Name "A_0005(ER1018-0001-0018)"}
	{attribute addProperty PreviousPort "A_0004(ER1008-0022-0017) : B"}
	A_0005_ER1018_0001_0018 : ER1018_78E8D3DD;
	{attribute addProperty Name "A_0006(ER1018-0002-0018)"}
	{attribute addProperty PreviousPort "A_0005(ER1018-0001-0018) : B"}
	A_0006_ER1018_0002_0018 : ER1018_78E8D3DD;
	{attribute addProperty Name "A_0007(ER1098-0001-0017)"}
	{attribute addProperty PreviousPort "A_0006(ER1018-0002-0018) : B"}
	A_0007_ER1098_0001_0017 : ER1098_78E8D3DD;
	{attribute addProperty Name "A_0008(ER1258-0001-0019)"}
	{attribute addProperty PreviousPort "A_0007(ER1098-0001-0017) : B"}
	A_0008_ER1258_0001_0019 : ER1258_58F475DD;
	{attribute addProperty Name "A_0009(ER1258-0001-0020)"}
	{attribute addProperty PreviousPort "A_0008(ER1258-0001-0019) : B"}
	A_0009_ER1258_0001_0020 : ER1258_58F475DD;
	{attribute addProperty Name "A_0010(ER1258-0002-0019)"}
	{attribute addProperty PreviousPort "A_0009(ER1258-0001-0020) : B"}
	A_0010_ER1258_0002_0019 : ER1258_58F475DD;
	{attribute addProperty Name "A_0011(ER1258-0002-0020)"}
	{attribute addProperty PreviousPort "A_0010(ER1258-0002-0019) : B"}
	A_0011_ER1258_0002_0020 : ER1258_58F475DD;
	{attribute addProperty Name "A_0012(ER1518-0002-0018)"}
	{attribute addProperty PreviousPort "A_0011(ER1258-0002-0020) : B"}
	A_0012_ER1518_0002_0018 : ER1518_CC442588;
	{attribute addProperty Name "A_0013(ER1518-0002-0019)"}
	{attribute addProperty PreviousPort "A_0012(ER1518-0002-0018) : B"}
	A_0013_ER1518_0002_0019 : ER1518_CC442588;
	{attribute addProperty Name "A_0014(ER1809-0021-0017)"}
	{attribute addProperty PreviousPort "A_0013(ER1518-0002-0019) : B"}
	A_0014_ER1809_0021_0017 : ER1809_32157CFD;
	{attribute addProperty Name "A_0015(ER1809-0022-0018)"}
	{attribute addProperty PreviousPort "A_0014(ER1809-0021-0017) : B"}
	A_0015_ER1809_0022_0018 : ER1809_32157CFD;
	{attribute addProperty Name "A_0016(ER1819-0021-0017)"}
	{attribute addProperty PreviousPort "A_0015(ER1809-0022-0018) : B"}
	A_0016_ER1819_0021_0017 : ER1819_32157CFD;
	{attribute addProperty Name "A_0017(ER1819-0022-0017)"}
	{attribute addProperty PreviousPort "A_0016(ER1819-0021-0017) : B"}
	A_0017_ER1819_0022_0017 : ER1819_32157CFD;
END_STRUCT
END_TYPE

// ---- DUTs/IO/Topology/Beckhoff_ER1xxx_A63E075A.TcDUT
{attribute 'GeneratedUsingTerminal: EK1100-0000-0018'}
{attribute addProperty BoxType "EK1100-0000-0018"}
{attribute addProperty Id "Beckhoff_ER1xxxEK1122Beckhoff_ER1xxxEK1122_4914C526508"}
{attribute addProperty CRC "2789082970"}
{attribute addProperty Size "508"}
{attribute addProperty Name "Beckhoff ER1xxx"}
TYPE Beckhoff_ER1xxx_A63E075A EXTENDS EK1100_1FC0878B :
STRUCT
	{attribute addProperty Name "Beckhoff ER1xxxEK1122"}
	{attribute addProperty PreviousPort "Beckhoff ER1xxx : B"}
	Beckhoff_ER1xxxEK1122 : Beckhoff_ER1xxxEK1122_4914C526;
END_STRUCT
END_TYPE

// ---- DUTs/IO/Topology/Beckhoff_ER2xxxEK1122_73471FC4.TcDUT
{attribute 'GeneratedUsingTerminal: EK1122-0000-0018'}
{attribute addProperty BoxType "EK1122-0000-0018"}
{attribute addProperty Id "Beckhoff_ER2xxxsub_EK1100EK1100_1FC0878B2A_0001_ER2008_0001_0018ER2008_E2806B9511A_0002_ER2008_0001_0019ER2008_E2806B9511A_0003_ER2008_0002_0018ER2008_E2806B9511A_0004_ER2008_0002_0019ER2008_E2806B9511A_0005_ER2008_0022_0017ER2008_E2806B9511A_0006_ER2008_0022_0018ER2008_E2806B9511A_0007_ER2028_0001_0017ER2028_E2806B9511A_0008_ER2028_0001_0018ER2028_E2806B9511A_0009_ER2028_0002_0018ER2028_E2806B9511A_0010_ER2028_0002_0019ER2028_E2806B9511A_0011_ER2028_1032_0016ER2028_E2806B9511A_0012_ER2038_0001_0017ER2038_3AE10DD720A_0013_ER2038_0001_0018ER2038_3AE10DD720A_0014_ER2038_0002_0017ER2038_3AE10DD720A_0015_ER2038_0002_0018ER2038_3AE10DD720A_0016_ER2308_0001_0018ER2308_F6D9A8D112A_0017_ER2308_0001_0019ER2308_F6D9A8D112A_0018_ER2308_0002_0018ER2308_F6D9A8D112A_0019_ER2308_0002_0019ER2308_F6D9A8D112A_0020_ER2318_0001_0018ER2318_F6D9A8D112A_0021_ER2318_0001_0019ER2318_F6D9A8D112A_0022_ER2318_0002_0018ER2318_F6D9A8D112A_0023_ER2318_0002_0019ER2318_F6D9A8D112A_0024_ER2328_0001_0017ER2328_F6D9A8D112A_0025_ER2328_0001_0018ER2328_F6D9A8D112A_0026_ER2328_0002_0018ER2328_F6D9A8D112A_0027_ER2328_0002_0019ER2328_F6D9A8D112A_0028_ER2338_0001_0022ER2338_7699BCF620A_0029_ER2338_0001_0023ER2338_7699BCF620A_0030_ER2338_0002_0022ER2338_7699BCF620A_0031_ER2338_0002_0023ER2338_7699BCF620A_0032_ER2338_1001_0017ER2338_7699BCF620A_0033_ER2338_1001_0018ER2338_7699BCF620A_0034_ER2338_1002_0017ER2338_7699BCF620A_0035_ER2338_1002_0018ER2338_7699BCF620A_0036_ER2339_0021_0018ER2339_D8E9F29A42A_0037_ER2339_0021_0019ER2339_4CF33DED36A_0038_ER2339_0022_0018ER2339_4CF33DED36A_0039_ER2339_0022_0019ER2339_4CF33DED36A_0040_ER2349_0021_0017ER2349_4CF33DED36A_0041_ER2349_0021_0018ER2349_4CF33DED36A_0042_ER2349_0022_0017ER2349_4CF33DED36A_0043_ER2349_0022_0018ER2349_4CF33DED36A_0044_ER2624_0002_0018ER2624_7B64371E7A_0045_ER2624_0002_0019ER2624_7B64371E7A_0046_ER2809_0021_0017ER2809_2B6483BD19A_0047_ER2809_0021_0018ER2809_2B6483BD19A_0048_ER2809_0022_0016ER2809_2B6483BD19A_0049_ER2809_0022_0017ER2809_2B6483BD19A_0050_ER2809_0022_0018ER2809_2B6483BD19"}
{attribute addProperty CRC "1934041028"}
{attribute addProperty Size "910"}
{attribute addProperty Name "Beckhoff ER2xxxEK1122"}
TYPE Beckhoff_ER2xxxEK1122_73471FC4 EXTENDS EK1122_1FC0878B :
STRUCT
	{attribute addProperty Name "Beckhoff ER2xxxsub EK1100"}
	{attribute addProperty PreviousPort "Beckhoff ER2xxxEK1122 : D"}
	Beckhoff_ER2xxxsub_EK1100 : EK1100_1FC0878B;
	{attribute addProperty Name "A_0001(ER2008-0001-0018)"}
	{attribute addProperty PreviousPort "Beckhoff ER2xxxsub EK1100 : C"}
	A_0001_ER2008_0001_0018 : ER2008_E2806B95;
	{attribute addProperty Name "A_0002(ER2008-0001-0019)"}
	{attribute addProperty PreviousPort "A_0001(ER2008-0001-0018) : B"}
	A_0002_ER2008_0001_0019 : ER2008_E2806B95;
	{attribute addProperty Name "A_0003(ER2008-0002-0018)"}
	{attribute addProperty PreviousPort "A_0002(ER2008-0001-0019) : B"}
	A_0003_ER2008_0002_0018 : ER2008_E2806B95;
	{attribute addProperty Name "A_0004(ER2008-0002-0019)"}
	{attribute addProperty PreviousPort "A_0003(ER2008-0002-0018) : B"}
	A_0004_ER2008_0002_0019 : ER2008_E2806B95;
	{attribute addProperty Name "A_0005(ER2008-0022-0017)"}
	{attribute addProperty PreviousPort "A_0004(ER2008-0002-0019) : B"}
	A_0005_ER2008_0022_0017 : ER2008_E2806B95;
	{attribute addProperty Name "A_0006(ER2008-0022-0018)"}
	{attribute addProperty PreviousPort "A_0005(ER2008-0022-0017) : B"}
	A_0006_ER2008_0022_0018 : ER2008_E2806B95;
	{attribute addProperty Name "A_0007(ER2028-0001-0017)"}
	{attribute addProperty PreviousPort "A_0006(ER2008-0022-0018) : B"}
	A_0007_ER2028_0001_0017 : ER2028_E2806B95;
	{attribute addProperty Name "A_0008(ER2028-0001-0018)"}
	{attribute addProperty PreviousPort "A_0007(ER2028-0001-0017) : B"}
	A_0008_ER2028_0001_0018 : ER2028_E2806B95;
	{attribute addProperty Name "A_0009(ER2028-0002-0018)"}
	{attribute addProperty PreviousPort "A_0008(ER2028-0001-0018) : B"}
	A_0009_ER2028_0002_0018 : ER2028_E2806B95;
	{attribute addProperty Name "A_0010(ER2028-0002-0019)"}
	{attribute addProperty PreviousPort "A_0009(ER2028-0002-0018) : B"}
	A_0010_ER2028_0002_0019 : ER2028_E2806B95;
	{attribute addProperty Name "A_0011(ER2028-1032-0016)"}
	{attribute addProperty PreviousPort "A_0010(ER2028-0002-0019) : B"}
	A_0011_ER2028_1032_0016 : ER2028_E2806B95;
	{attribute addProperty Name "A_0012(ER2038-0001-0017)"}
	{attribute addProperty PreviousPort "A_0011(ER2028-1032-0016) : B"}
	A_0012_ER2038_0001_0017 : ER2038_3AE10DD7;
	{attribute addProperty Name "A_0013(ER2038-0001-0018)"}
	{attribute addProperty PreviousPort "A_0012(ER2038-0001-0017) : B"}
	A_0013_ER2038_0001_0018 : ER2038_3AE10DD7;
	{attribute addProperty Name "A_0014(ER2038-0002-0017)"}
	{attribute addProperty PreviousPort "A_0013(ER2038-0001-0018) : B"}
	A_0014_ER2038_0002_0017 : ER2038_3AE10DD7;
	{attribute addProperty Name "A_0015(ER2038-0002-0018)"}
	{attribute addProperty PreviousPort "A_0014(ER2038-0002-0017) : B"}
	A_0015_ER2038_0002_0018 : ER2038_3AE10DD7;
	{attribute addProperty Name "A_0016(ER2308-0001-0018)"}
	{attribute addProperty PreviousPort "A_0015(ER2038-0002-0018) : B"}
	A_0016_ER2308_0001_0018 : ER2308_F6D9A8D1;
	{attribute addProperty Name "A_0017(ER2308-0001-0019)"}
	{attribute addProperty PreviousPort "A_0016(ER2308-0001-0018) : B"}
	A_0017_ER2308_0001_0019 : ER2308_F6D9A8D1;
	{attribute addProperty Name "A_0018(ER2308-0002-0018)"}
	{attribute addProperty PreviousPort "A_0017(ER2308-0001-0019) : B"}
	A_0018_ER2308_0002_0018 : ER2308_F6D9A8D1;
	{attribute addProperty Name "A_0019(ER2308-0002-0019)"}
	{attribute addProperty PreviousPort "A_0018(ER2308-0002-0018) : B"}
	A_0019_ER2308_0002_0019 : ER2308_F6D9A8D1;
	{attribute addProperty Name "A_0020(ER2318-0001-0018)"}
	{attribute addProperty PreviousPort "A_0019(ER2308-0002-0019) : B"}
	A_0020_ER2318_0001_0018 : ER2318_F6D9A8D1;
	{attribute addProperty Name "A_0021(ER2318-0001-0019)"}
	{attribute addProperty PreviousPort "A_0020(ER2318-0001-0018) : B"}
	A_0021_ER2318_0001_0019 : ER2318_F6D9A8D1;
	{attribute addProperty Name "A_0022(ER2318-0002-0018)"}
	{attribute addProperty PreviousPort "A_0021(ER2318-0001-0019) : B"}
	A_0022_ER2318_0002_0018 : ER2318_F6D9A8D1;
	{attribute addProperty Name "A_0023(ER2318-0002-0019)"}
	{attribute addProperty PreviousPort "A_0022(ER2318-0002-0018) : B"}
	A_0023_ER2318_0002_0019 : ER2318_F6D9A8D1;
	{attribute addProperty Name "A_0024(ER2328-0001-0017)"}
	{attribute addProperty PreviousPort "A_0023(ER2318-0002-0019) : B"}
	A_0024_ER2328_0001_0017 : ER2328_F6D9A8D1;
	{attribute addProperty Name "A_0025(ER2328-0001-0018)"}
	{attribute addProperty PreviousPort "A_0024(ER2328-0001-0017) : B"}
	A_0025_ER2328_0001_0018 : ER2328_F6D9A8D1;
	{attribute addProperty Name "A_0026(ER2328-0002-0018)"}
	{attribute addProperty PreviousPort "A_0025(ER2328-0001-0018) : B"}
	A_0026_ER2328_0002_0018 : ER2328_F6D9A8D1;
	{attribute addProperty Name "A_0027(ER2328-0002-0019)"}
	{attribute addProperty PreviousPort "A_0026(ER2328-0002-0018) : B"}
	A_0027_ER2328_0002_0019 : ER2328_F6D9A8D1;
	{attribute addProperty Name "A_0028(ER2338-0001-0022)"}
	{attribute addProperty PreviousPort "A_0027(ER2328-0002-0019) : B"}
	A_0028_ER2338_0001_0022 : ER2338_7699BCF6;
	{attribute addProperty Name "A_0029(ER2338-0001-0023)"}
	{attribute addProperty PreviousPort "A_0028(ER2338-0001-0022) : B"}
	A_0029_ER2338_0001_0023 : ER2338_7699BCF6;
	{attribute addProperty Name "A_0030(ER2338-0002-0022)"}
	{attribute addProperty PreviousPort "A_0029(ER2338-0001-0023) : B"}
	A_0030_ER2338_0002_0022 : ER2338_7699BCF6;
	{attribute addProperty Name "A_0031(ER2338-0002-0023)"}
	{attribute addProperty PreviousPort "A_0030(ER2338-0002-0022) : B"}
	A_0031_ER2338_0002_0023 : ER2338_7699BCF6;
	{attribute addProperty Name "A_0032(ER2338-1001-0017)"}
	{attribute addProperty PreviousPort "A_0031(ER2338-0002-0023) : B"}
	A_0032_ER2338_1001_0017 : ER2338_7699BCF6;
	{attribute addProperty Name "A_0033(ER2338-1001-0018)"}
	{attribute addProperty PreviousPort "A_0032(ER2338-1001-0017) : B"}
	A_0033_ER2338_1001_0018 : ER2338_7699BCF6;
	{attribute addProperty Name "A_0034(ER2338-1002-0017)"}
	{attribute addProperty PreviousPort "A_0033(ER2338-1001-0018) : B"}
	A_0034_ER2338_1002_0017 : ER2338_7699BCF6;
	{attribute addProperty Name "A_0035(ER2338-1002-0018)"}
	{attribute addProperty PreviousPort "A_0034(ER2338-1002-0017) : B"}
	A_0035_ER2338_1002_0018 : ER2338_7699BCF6;
	{attribute addProperty Name "A_0036(ER2339-0021-0018)"}
	{attribute addProperty PreviousPort "A_0035(ER2338-1002-0018) : B"}
	A_0036_ER2339_0021_0018 : ER2339_D8E9F29A;
	{attribute addProperty Name "A_0037(ER2339-0021-0019)"}
	{attribute addProperty PreviousPort "A_0036(ER2339-0021-0018) : B"}
	A_0037_ER2339_0021_0019 : ER2339_4CF33DED;
	{attribute addProperty Name "A_0038(ER2339-0022-0018)"}
	{attribute addProperty PreviousPort "A_0037(ER2339-0021-0019) : B"}
	A_0038_ER2339_0022_0018 : ER2339_4CF33DED;
	{attribute addProperty Name "A_0039(ER2339-0022-0019)"}
	{attribute addProperty PreviousPort "A_0038(ER2339-0022-0018) : B"}
	A_0039_ER2339_0022_0019 : ER2339_4CF33DED;
	{attribute addProperty Name "A_0040(ER2349-0021-0017)"}
	{attribute addProperty PreviousPort "A_0039(ER2339-0022-0019) : B"}
	A_0040_ER2349_0021_0017 : ER2349_4CF33DED;
	{attribute addProperty Name "A_0041(ER2349-0021-0018)"}
	{attribute addProperty PreviousPort "A_0040(ER2349-0021-0017) : B"}
	A_0041_ER2349_0021_0018 : ER2349_4CF33DED;
	{attribute addProperty Name "A_0042(ER2349-0022-0017)"}
	{attribute addProperty PreviousPort "A_0041(ER2349-0021-0018) : B"}
	A_0042_ER2349_0022_0017 : ER2349_4CF33DED;
	{attribute addProperty Name "A_0043(ER2349-0022-0018)"}
	{attribute addProperty PreviousPort "A_0042(ER2349-0022-0017) : B"}
	A_0043_ER2349_0022_0018 : ER2349_4CF33DED;
	{attribute addProperty Name "A_0044(ER2624-0002-0018)"}
	{attribute addProperty PreviousPort "A_0043(ER2349-0022-0018) : B"}
	A_0044_ER2624_0002_0018 : ER2624_7B64371E;
	{attribute addProperty Name "A_0045(ER2624-0002-0019)"}
	{attribute addProperty PreviousPort "A_0044(ER2624-0002-0018) : B"}
	A_0045_ER2624_0002_0019 : ER2624_7B64371E;
	{attribute addProperty Name "A_0046(ER2809-0021-0017)"}
	{attribute addProperty PreviousPort "A_0045(ER2624-0002-0019) : B"}
	A_0046_ER2809_0021_0017 : ER2809_2B6483BD;
	{attribute addProperty Name "A_0047(ER2809-0021-0018)"}
	{attribute addProperty PreviousPort "A_0046(ER2809-0021-0017) : B"}
	A_0047_ER2809_0021_0018 : ER2809_2B6483BD;
	{attribute addProperty Name "A_0048(ER2809-0022-0016)"}
	{attribute addProperty PreviousPort "A_0047(ER2809-0021-0018) : B"}
	A_0048_ER2809_0022_0016 : ER2809_2B6483BD;
	{attribute addProperty Name "A_0049(ER2809-0022-0017)"}
	{attribute addProperty PreviousPort "A_0048(ER2809-0022-0016) : B"}
	A_0049_ER2809_0022_0017 : ER2809_2B6483BD;
	{attribute addProperty Name "A_0050(ER2809-0022-0018)"}
	{attribute addProperty PreviousPort "A_0049(ER2809-0022-0017) : B"}
	A_0050_ER2809_0022_0018 : ER2809_2B6483BD;
END_STRUCT
END_TYPE

// ---- DUTs/IO/Topology/Beckhoff_ER2xxx_CED8BB26.TcDUT
{attribute 'GeneratedUsingTerminal: EK1100-0000-0018'}
{attribute addProperty BoxType "EK1100-0000-0018"}
{attribute addProperty Id "Beckhoff_ER2xxxEK1122Beckhoff_ER2xxxEK1122_73471FC4910"}
{attribute addProperty CRC "3470310182"}
{attribute addProperty Size "910"}
{attribute addProperty Name "Beckhoff ER2xxx"}
TYPE Beckhoff_ER2xxx_CED8BB26 EXTENDS EK1100_1FC0878B :
STRUCT
	{attribute addProperty Name "Beckhoff ER2xxxEK1122"}
	{attribute addProperty PreviousPort "Beckhoff ER2xxx : B"}
	Beckhoff_ER2xxxEK1122 : Beckhoff_ER2xxxEK1122_73471FC4;
END_STRUCT
END_TYPE

// ---- DUTs/IO/Topology/Beckhoff_ER3xxxEK1122_4F8E32D9.TcDUT
{attribute 'GeneratedUsingTerminal: EK1122-0000-0018'}
{attribute addProperty BoxType "EK1122-0000-0018"}
{attribute addProperty Id "Beckhoff_ER3xxxsub_EK1100EK1100_1FC0878B2A_0001_ER3174_0002_0016ER3174_DCC7866252A_0002_ER3174_0002_0022ER3174_DCC7866252A_0003_ER3174_0002_0023ER3174_DCC7866252A_0004_ER3184_0002_0019ER3184_DCC7866252A_0005_ER3184_0002_0020ER3184_DCC7866252A_0006_ER3184_0002_0021ER3184_DCC7866252A_0007_ER3184_1002_0020ER3184_DCC7866252A_0008_ER3184_1002_0021ER3184_DCC7866252A_0009_ER3204_0002_0016ER3204_6CD7E11952A_0010_ER3204_0002_0020ER3204_6CD7E11952A_0011_ER3204_0002_0021ER3204_AB25C3AC48A_0012_ER3314_0002_0021ER3314_E65CDB1C48"}
{attribute addProperty CRC "1334719193"}
{attribute addProperty Size "618"}
{attribute addProperty Name "Beckhoff ER3xxxEK1122"}
TYPE Beckhoff_ER3xxxEK1122_4F8E32D9 EXTENDS EK1122_1FC0878B :
STRUCT
	{attribute addProperty Name "Beckhoff ER3xxxsub EK1100"}
	{attribute addProperty PreviousPort "Beckhoff ER3xxxEK1122 : D"}
	Beckhoff_ER3xxxsub_EK1100 : EK1100_1FC0878B;
	{attribute addProperty Name "A_0001(ER3174-0002-0016)"}
	{attribute addProperty PreviousPort "Beckhoff ER3xxxsub EK1100 : C"}
	A_0001_ER3174_0002_0016 : ER3174_DCC78662;
	{attribute addProperty Name "A_0002(ER3174-0002-0022)"}
	{attribute addProperty PreviousPort "A_0001(ER3174-0002-0016) : B"}
	A_0002_ER3174_0002_0022 : ER3174_DCC78662;
	{attribute addProperty Name "A_0003(ER3174-0002-0023)"}
	{attribute addProperty PreviousPort "A_0002(ER3174-0002-0022) : B"}
	A_0003_ER3174_0002_0023 : ER3174_DCC78662;
	{attribute addProperty Name "A_0004(ER3184-0002-0019)"}
	{attribute addProperty PreviousPort "A_0003(ER3174-0002-0023) : B"}
	A_0004_ER3184_0002_0019 : ER3184_DCC78662;
	{attribute addProperty Name "A_0005(ER3184-0002-0020)"}
	{attribute addProperty PreviousPort "A_0004(ER3184-0002-0019) : B"}
	A_0005_ER3184_0002_0020 : ER3184_DCC78662;
	{attribute addProperty Name "A_0006(ER3184-0002-0021)"}
	{attribute addProperty PreviousPort "A_0005(ER3184-0002-0020) : B"}
	A_0006_ER3184_0002_0021 : ER3184_DCC78662;
	{attribute addProperty Name "A_0007(ER3184-1002-0020)"}
	{attribute addProperty PreviousPort "A_0006(ER3184-0002-0021) : B"}
	A_0007_ER3184_1002_0020 : ER3184_DCC78662;
	{attribute addProperty Name "A_0008(ER3184-1002-0021)"}
	{attribute addProperty PreviousPort "A_0007(ER3184-1002-0020) : B"}
	A_0008_ER3184_1002_0021 : ER3184_DCC78662;
	{attribute addProperty Name "A_0009(ER3204-0002-0016)"}
	{attribute addProperty PreviousPort "A_0008(ER3184-1002-0021) : B"}
	A_0009_ER3204_0002_0016 : ER3204_6CD7E119;
	{attribute addProperty Name "A_0010(ER3204-0002-0020)"}
	{attribute addProperty PreviousPort "A_0009(ER3204-0002-0016) : B"}
	A_0010_ER3204_0002_0020 : ER3204_6CD7E119;
	{attribute addProperty Name "A_0011(ER3204-0002-0021)"}
	{attribute addProperty PreviousPort "A_0010(ER3204-0002-0020) : B"}
	A_0011_ER3204_0002_0021 : ER3204_AB25C3AC;
	{attribute addProperty Name "A_0012(ER3314-0002-0021)"}
	{attribute addProperty PreviousPort "A_0011(ER3204-0002-0021) : B"}
	A_0012_ER3314_0002_0021 : ER3314_E65CDB1C;
END_STRUCT
END_TYPE

// ---- DUTs/IO/Topology/Beckhoff_ER3xxx_58A653D9.TcDUT
{attribute 'GeneratedUsingTerminal: EK1100-0000-0018'}
{attribute addProperty BoxType "EK1100-0000-0018"}
{attribute addProperty Id "Beckhoff_ER3xxxEK1122Beckhoff_ER3xxxEK1122_4F8E32D9618"}
{attribute addProperty CRC "1487295449"}
{attribute addProperty Size "618"}
{attribute addProperty Name "Beckhoff ER3xxx"}
TYPE Beckhoff_ER3xxx_58A653D9 EXTENDS EK1100_1FC0878B :
STRUCT
	{attribute addProperty Name "Beckhoff ER3xxxEK1122"}
	{attribute addProperty PreviousPort "Beckhoff ER3xxx : B"}
	Beckhoff_ER3xxxEK1122 : Beckhoff_ER3xxxEK1122_4F8E32D9;
END_STRUCT
END_TYPE

// ---- DUTs/IO/Topology/Beckhoff_ER4xxxEK1122_5C895096.TcDUT
{attribute 'GeneratedUsingTerminal: EK1122-0000-0018'}
{attribute addProperty BoxType "EK1122-0000-0018"}
{attribute addProperty Id "Beckhoff_ER4xxxsub_EK1100EK1100_1FC0878B2A_0001_ER4174_0002_0016ER4174_AB92710E19A_0002_ER4174_0002_0019ER4174_AB92710E19A_0003_ER4374_0002_0018ER4374_A304750F36A_0004_ER4374_0002_0019ER4374_A304750F36"}
{attribute addProperty CRC "1552502934"}
{attribute addProperty Size "112"}
{attribute addProperty Name "Beckhoff ER4xxxEK1122"}
TYPE Beckhoff_ER4xxxEK1122_5C895096 EXTENDS EK1122_1FC0878B :
STRUCT
	{attribute addProperty Name "Beckhoff ER4xxxsub EK1100"}
	{attribute addProperty PreviousPort "Beckhoff ER4xxxEK1122 : D"}
	Beckhoff_ER4xxxsub_EK1100 : EK1100_1FC0878B;
	{attribute addProperty Name "A_0001(ER4174-0002-0016)"}
	{attribute addProperty PreviousPort "Beckhoff ER4xxxsub EK1100 : C"}
	A_0001_ER4174_0002_0016 : ER4174_AB92710E;
	{attribute addProperty Name "A_0002(ER4174-0002-0019)"}
	{attribute addProperty PreviousPort "A_0001(ER4174-0002-0016) : B"}
	A_0002_ER4174_0002_0019 : ER4174_AB92710E;
	{attribute addProperty Name "A_0003(ER4374-0002-0018)"}
	{attribute addProperty PreviousPort "A_0002(ER4174-0002-0019) : B"}
	A_0003_ER4374_0002_0018 : ER4374_A304750F;
	{attribute addProperty Name "A_0004(ER4374-0002-0019)"}
	{attribute addProperty PreviousPort "A_0003(ER4374-0002-0018) : B"}
	A_0004_ER4374_0002_0019 : ER4374_A304750F;
END_STRUCT
END_TYPE

// ---- DUTs/IO/Topology/Beckhoff_ER4xxx_797AEBB5.TcDUT
{attribute 'GeneratedUsingTerminal: EK1100-0000-0018'}
{attribute addProperty BoxType "EK1100-0000-0018"}
{attribute addProperty Id "Beckhoff_ER4xxxEK1122Beckhoff_ER4xxxEK1122_5C895096112"}
{attribute addProperty CRC "2038098869"}
{attribute addProperty Size "112"}
{attribute addProperty Name "Beckhoff ER4xxx"}
TYPE Beckhoff_ER4xxx_797AEBB5 EXTENDS EK1100_1FC0878B :
STRUCT
	{attribute addProperty Name "Beckhoff ER4xxxEK1122"}
	{attribute addProperty PreviousPort "Beckhoff ER4xxx : B"}
	Beckhoff_ER4xxxEK1122 : Beckhoff_ER4xxxEK1122_5C895096;
END_STRUCT
END_TYPE

// ---- DUTs/IO/Topology/Beckhoff_ER5xxxEK1122_B89AF081.TcDUT
{attribute 'GeneratedUsingTerminal: EK1122-0000-0018'}
{attribute addProperty BoxType "EK1122-0000-0018"}
{attribute addProperty Id "Beckhoff_ER5xxxsub_EK1100EK1100_1FC0878B2A_0001_ER5101_0002_0019ER5101_87AC78CF32A_0002_ER5101_1002_0017ER5101_87AC78CF32A_0003_ER5151_0002_0018ER5151_7476E94838"}
{attribute addProperty CRC "3097161857"}
{attribute addProperty Size "104"}
{attribute addProperty Name "Beckhoff ER5xxxEK1122"}
TYPE Beckhoff_ER5xxxEK1122_B89AF081 EXTENDS EK1122_1FC0878B :
STRUCT
	{attribute addProperty Name "Beckhoff ER5xxxsub EK1100"}
	{attribute addProperty PreviousPort "Beckhoff ER5xxxEK1122 : D"}
	Beckhoff_ER5xxxsub_EK1100 : EK1100_1FC0878B;
	{attribute addProperty Name "A_0001(ER5101-0002-0019)"}
	{attribute addProperty PreviousPort "Beckhoff ER5xxxsub EK1100 : C"}
	A_0001_ER5101_0002_0019 : ER5101_87AC78CF;
	{attribute addProperty Name "A_0002(ER5101-1002-0017)"}
	{attribute addProperty PreviousPort "A_0001(ER5101-0002-0019) : B"}
	A_0002_ER5101_1002_0017 : ER5101_87AC78CF;
	{attribute addProperty Name "A_0003(ER5151-0002-0018)"}
	{attribute addProperty PreviousPort "A_0002(ER5101-1002-0017) : B"}
	A_0003_ER5151_0002_0018 : ER5151_7476E948;
END_STRUCT
END_TYPE

// ---- DUTs/IO/Topology/Beckhoff_ER5xxx_22A4CB20.TcDUT
{attribute 'GeneratedUsingTerminal: EK1100-0000-0018'}
{attribute addProperty BoxType "EK1100-0000-0018"}
{attribute addProperty Id "Beckhoff_ER5xxxEK1122Beckhoff_ER5xxxEK1122_B89AF081104"}
{attribute addProperty CRC "581225248"}
{attribute addProperty Size "104"}
{attribute addProperty Name "Beckhoff ER5xxx"}
TYPE Beckhoff_ER5xxx_22A4CB20 EXTENDS EK1100_1FC0878B :
STRUCT
	{attribute addProperty Name "Beckhoff ER5xxxEK1122"}
	{attribute addProperty PreviousPort "Beckhoff ER5xxx : B"}
	Beckhoff_ER5xxxEK1122 : Beckhoff_ER5xxxEK1122_B89AF081;
END_STRUCT
END_TYPE

// ---- DUTs/IO/Topology/Beckhoff_ER6xxxEK1122_BD5112F1.TcDUT
{attribute 'GeneratedUsingTerminal: EK1122-0000-0018'}
{attribute addProperty BoxType "EK1122-0000-0018"}
{attribute addProperty Id "Beckhoff_ER6xxxsub_EK1100EK1100_1FC0878B2A_0001_ER6001_0002_0016ER6001_40883D0360A_0002_ER6001_0002_0021ER6001_40883D0360A_0003_ER6002_0002_0021ER6002_7F53816A108A_0004_ER6002_0002_0022ER6002_7BE6B617108A_0005_ER6002_0002_0023ER6002_7BE6B617108"}
{attribute addProperty CRC "3176207089"}
{attribute addProperty Size "446"}
{attribute addProperty Name "Beckhoff ER6xxxEK1122"}
TYPE Beckhoff_ER6xxxEK1122_BD5112F1 EXTENDS EK1122_1FC0878B :
STRUCT
	{attribute addProperty Name "Beckhoff ER6xxxsub EK1100"}
	{attribute addProperty PreviousPort "Beckhoff ER6xxxEK1122 : D"}
	Beckhoff_ER6xxxsub_EK1100 : EK1100_1FC0878B;
	{attribute addProperty Name "A_0001(ER6001-0002-0016)"}
	{attribute addProperty PreviousPort "Beckhoff ER6xxxsub EK1100 : C"}
	A_0001_ER6001_0002_0016 : ER6001_40883D03;
	{attribute addProperty Name "A_0002(ER6001-0002-0021)"}
	{attribute addProperty PreviousPort "A_0001(ER6001-0002-0016) : B"}
	A_0002_ER6001_0002_0021 : ER6001_40883D03;
	{attribute addProperty Name "A_0003(ER6002-0002-0021)"}
	{attribute addProperty PreviousPort "A_0002(ER6001-0002-0021) : B"}
	A_0003_ER6002_0002_0021 : ER6002_7F53816A;
	{attribute addProperty Name "A_0004(ER6002-0002-0022)"}
	{attribute addProperty PreviousPort "A_0003(ER6002-0002-0021) : B"}
	A_0004_ER6002_0002_0022 : ER6002_7BE6B617;
	{attribute addProperty Name "A_0005(ER6002-0002-0023)"}
	{attribute addProperty PreviousPort "A_0004(ER6002-0002-0022) : B"}
	A_0005_ER6002_0002_0023 : ER6002_7BE6B617;
END_STRUCT
END_TYPE

// ---- DUTs/IO/Topology/Beckhoff_ER6xxx_896D799E.TcDUT
{attribute 'GeneratedUsingTerminal: EK1100-0000-0018'}
{attribute addProperty BoxType "EK1100-0000-0018"}
{attribute addProperty Id "Beckhoff_ER6xxxEK1122Beckhoff_ER6xxxEK1122_BD5112F1446"}
{attribute addProperty CRC "2305653150"}
{attribute addProperty Size "446"}
{attribute addProperty Name "Beckhoff ER6xxx"}
TYPE Beckhoff_ER6xxx_896D799E EXTENDS EK1100_1FC0878B :
STRUCT
	{attribute addProperty Name "Beckhoff ER6xxxEK1122"}
	{attribute addProperty PreviousPort "Beckhoff ER6xxx : B"}
	Beckhoff_ER6xxxEK1122 : Beckhoff_ER6xxxEK1122_BD5112F1;
END_STRUCT
END_TYPE

// ---- DUTs/IO/Topology/Beckhoff_ER7xxxEK1122_0EBE6E72.TcDUT
{attribute 'GeneratedUsingTerminal: EK1122-0000-0018'}
{attribute addProperty BoxType "EK1122-0000-0018"}
{attribute addProperty Id "Beckhoff_ER7xxxsub_EK1100EK1100_1FC0878B2A_0001_ER7041_0002_0024ER7041_3210CF4053A_0002_ER7041_0002_0025ER7041_3210CF4053A_0003_ER7041_1002_0024ER7041_3210CF4053A_0004_ER7041_1002_0025ER7041_3210CF4053A_0005_ER7041_2002_0024ER7041_3210CF4053A_0006_ER7041_2002_0025ER7041_3210CF4053A_0007_ER7041_3002_0021ER7041_3E4BEAEF54A_0008_ER7041_3002_0022ER7041_3E4BEAEF54A_0009_ER7342_0002_0020ER7342_2AE9C6B386A_0010_ER7342_0002_0021ER7342_2AE9C6B386A_0011_ER7342_0002_0022ER7342_2AE9C6B386"}
{attribute addProperty CRC "247361138"}
{attribute addProperty Size "686"}
{attribute addProperty Name "Beckhoff ER7xxxEK1122"}
TYPE Beckhoff_ER7xxxEK1122_0EBE6E72 EXTENDS EK1122_1FC0878B :
STRUCT
	{attribute addProperty Name "Beckhoff ER7xxxsub EK1100"}
	{attribute addProperty PreviousPort "Beckhoff ER7xxxEK1122 : D"}
	Beckhoff_ER7xxxsub_EK1100 : EK1100_1FC0878B;
	{attribute addProperty Name "A_0001(ER7041-0002-0024)"}
	{attribute addProperty PreviousPort "Beckhoff ER7xxxsub EK1100 : C"}
	A_0001_ER7041_0002_0024 : ER7041_3210CF40;
	{attribute addProperty Name "A_0002(ER7041-0002-0025)"}
	{attribute addProperty PreviousPort "A_0001(ER7041-0002-0024) : B"}
	A_0002_ER7041_0002_0025 : ER7041_3210CF40;
	{attribute addProperty Name "A_0003(ER7041-1002-0024)"}
	{attribute addProperty PreviousPort "A_0002(ER7041-0002-0025) : B"}
	A_0003_ER7041_1002_0024 : ER7041_3210CF40;
	{attribute addProperty Name "A_0004(ER7041-1002-0025)"}
	{attribute addProperty PreviousPort "A_0003(ER7041-1002-0024) : B"}
	A_0004_ER7041_1002_0025 : ER7041_3210CF40;
	{attribute addProperty Name "A_0005(ER7041-2002-0024)"}
	{attribute addProperty PreviousPort "A_0004(ER7041-1002-0025) : B"}
	A_0005_ER7041_2002_0024 : ER7041_3210CF40;
	{attribute addProperty Name "A_0006(ER7041-2002-0025)"}
	{attribute addProperty PreviousPort "A_0005(ER7041-2002-0024) : B"}
	A_0006_ER7041_2002_0025 : ER7041_3210CF40;
	{attribute addProperty Name "A_0007(ER7041-3002-0021)"}
	{attribute addProperty PreviousPort "A_0006(ER7041-2002-0025) : B"}
	A_0007_ER7041_3002_0021 : ER7041_3E4BEAEF;
	{attribute addProperty Name "A_0008(ER7041-3002-0022)"}
	{attribute addProperty PreviousPort "A_0007(ER7041-3002-0021) : B"}
	A_0008_ER7041_3002_0022 : ER7041_3E4BEAEF;
	{attribute addProperty Name "A_0009(ER7342-0002-0020)"}
	{attribute addProperty PreviousPort "A_0008(ER7041-3002-0022) : B"}
	A_0009_ER7342_0002_0020 : ER7342_2AE9C6B3;
	{attribute addProperty Name "A_0010(ER7342-0002-0021)"}
	{attribute addProperty PreviousPort "A_0009(ER7342-0002-0020) : B"}
	A_0010_ER7342_0002_0021 : ER7342_2AE9C6B3;
	{attribute addProperty Name "A_0011(ER7342-0002-0022)"}
	{attribute addProperty PreviousPort "A_0010(ER7342-0002-0021) : B"}
	A_0011_ER7342_0002_0022 : ER7342_2AE9C6B3;
END_STRUCT
END_TYPE

// ---- DUTs/IO/Topology/Beckhoff_ER7xxx_FFC5AE47.TcDUT
{attribute 'GeneratedUsingTerminal: EK1100-0000-0018'}
{attribute addProperty BoxType "EK1100-0000-0018"}
{attribute addProperty Id "Beckhoff_ER7xxxEK1122Beckhoff_ER7xxxEK1122_0EBE6E72686"}
{attribute addProperty CRC "4291145287"}
{attribute addProperty Size "686"}
{attribute addProperty Name "Beckhoff ER7xxx"}
TYPE Beckhoff_ER7xxx_FFC5AE47 EXTENDS EK1100_1FC0878B :
STRUCT
	{attribute addProperty Name "Beckhoff ER7xxxEK1122"}
	{attribute addProperty PreviousPort "Beckhoff ER7xxx : B"}
	Beckhoff_ER7xxxEK1122 : Beckhoff_ER7xxxEK1122_0EBE6E72;
END_STRUCT
END_TYPE

// ---- DUTs/IO/Topology/Beckhoff_ER8xxxEK1122_CCFAC454.TcDUT
{attribute 'GeneratedUsingTerminal: EK1122-0000-0018'}
{attribute addProperty BoxType "EK1122-0000-0018"}
{attribute addProperty Id "Beckhoff_ER8xxxsub_EK1100EK1100_1FC0878B2A_0001_ER8309_1022_0018ER8309_A0C54F7770"}
{attribute addProperty CRC "3438986324"}
{attribute addProperty Size "72"}
{attribute addProperty Name "Beckhoff ER8xxxEK1122"}
TYPE Beckhoff_ER8xxxEK1122_CCFAC454 EXTENDS EK1122_1FC0878B :
STRUCT
	{attribute addProperty Name "Beckhoff ER8xxxsub EK1100"}
	{attribute addProperty PreviousPort "Beckhoff ER8xxxEK1122 : D"}
	Beckhoff_ER8xxxsub_EK1100 : EK1100_1FC0878B;
	{attribute addProperty Name "A_0001(ER8309-1022-0018)"}
	{attribute addProperty PreviousPort "Beckhoff ER8xxxsub EK1100 : C"}
	A_0001_ER8309_1022_0018 : ER8309_A0C54F77;
END_STRUCT
END_TYPE

// ---- DUTs/IO/Topology/Beckhoff_ER8xxx_509945A9.TcDUT
{attribute 'GeneratedUsingTerminal: EK1100-0000-0018'}
{attribute addProperty BoxType "EK1100-0000-0018"}
{attribute addProperty Id "Beckhoff_ER8xxxEK1122Beckhoff_ER8xxxEK1122_CCFAC45472"}
{attribute addProperty CRC "1352222121"}
{attribute addProperty Size "72"}
{attribute addProperty Name "Beckhoff ER8xxx"}
TYPE Beckhoff_ER8xxx_509945A9 EXTENDS EK1100_1FC0878B :
STRUCT
	{attribute addProperty Name "Beckhoff ER8xxxEK1122"}
	{attribute addProperty PreviousPort "Beckhoff ER8xxx : B"}
	Beckhoff_ER8xxxEK1122 : Beckhoff_ER8xxxEK1122_CCFAC454;
END_STRUCT
END_TYPE

// ---- DUTs/IO/Topology/EtherCAT_Master_ERxxxx_879C9A05.TcDUT
{attribute 'GeneratedUsingTerminal: IODEVICETYPE_ETHERCATPROT'}
{attribute addProperty BoxType "IODEVICETYPE_ETHERCATPROT"}
{attribute addProperty Id "Beckhoff_ER1xxxBeckhoff_ER1xxx_A63E075A508Beckhoff_ER2xxxBeckhoff_ER2xxx_CED8BB26910Beckhoff_ER3xxxBeckhoff_ER3xxx_58A653D9618Beckhoff_ER4xxxBeckhoff_ER4xxx_797AEBB5112Beckhoff_ER5xxxBeckhoff_ER5xxx_22A4CB20104Beckhoff_ER6xxxBeckhoff_ER6xxx_896D799E446Beckhoff_ER7xxxBeckhoff_ER7xxx_FFC5AE47686Beckhoff_ER8xxxBeckhoff_ER8xxx_509945A972SyncUnitsSyncUnits_99E584AF18InputsInputs_25A0042B160OutputsOutputs_2397A10E106InfoDataInfoData_E68C61CD28"}
{attribute addProperty CRC "2275187205"}
{attribute addProperty Size "3768"}
{attribute addProperty Name "EtherCAT Master ERxxxx"}
TYPE EtherCAT_Master_ERxxxx_879C9A05 EXTENDS EtcMasterBase_62654B43 :
STRUCT
	{attribute addProperty Name "Beckhoff ER1xxx"}
	{attribute addProperty PreviousPort "EtherCAT Master ERxxxx : Master"}
	Beckhoff_ER1xxx : Beckhoff_ER1xxx_A63E075A;
	{attribute addProperty Name "Beckhoff ER2xxx"}
	{attribute addProperty PreviousPort "Beckhoff ER1xxx : C"}
	Beckhoff_ER2xxx : Beckhoff_ER2xxx_CED8BB26;
	{attribute addProperty Name "Beckhoff ER3xxx"}
	{attribute addProperty PreviousPort "Beckhoff ER2xxx : C"}
	Beckhoff_ER3xxx : Beckhoff_ER3xxx_58A653D9;
	{attribute addProperty Name "Beckhoff ER4xxx"}
	{attribute addProperty PreviousPort "Beckhoff ER3xxx : C"}
	Beckhoff_ER4xxx : Beckhoff_ER4xxx_797AEBB5;
	{attribute addProperty Name "Beckhoff ER5xxx"}
	{attribute addProperty PreviousPort "Beckhoff ER4xxx : C"}
	Beckhoff_ER5xxx : Beckhoff_ER5xxx_22A4CB20;
	{attribute addProperty Name "Beckhoff ER6xxx"}
	{attribute addProperty PreviousPort "Beckhoff ER5xxx : C"}
	Beckhoff_ER6xxx : Beckhoff_ER6xxx_896D799E;
	{attribute addProperty Name "Beckhoff ER7xxx"}
	{attribute addProperty PreviousPort "Beckhoff ER6xxx : C"}
	Beckhoff_ER7xxx : Beckhoff_ER7xxx_FFC5AE47;
	{attribute addProperty Name "Beckhoff ER8xxx"}
	{attribute addProperty PreviousPort "Beckhoff ER7xxx : C"}
	Beckhoff_ER8xxx : Beckhoff_ER8xxx_509945A9;
	{attribute addProperty Name "SyncUnits"}
	SyncUnits : SyncUnits_99E584AF;
	{attribute addProperty Name "Inputs"}
	Inputs : Inputs_25A0042B;
	{attribute addProperty Name "Outputs"}
	Outputs : Outputs_2397A10E;
	{attribute addProperty Name "InfoData"}
	InfoData : InfoData_E68C61CD;
END_STRUCT
END_TYPE

// ---- DUTs/IO/Base/EtcSlaveBase_82538BE2.TcDUT

TYPE EtcSlaveBase_82538BE2 :
STRUCT
END_STRUCT
END_TYPE

// ---- DUTs/IO/Base/EtcSlaveBase_82538BE2.TcDUT

TYPE EtcSlaveBase_82538BE2 :
STRUCT
END_STRUCT
END_TYPE

// ---- DUTs/IO/Base/EtcSlaveBase_82538BE2.TcDUT

TYPE EtcSlaveBase_82538BE2 :
STRUCT
END_STRUCT
END_TYPE

// ---- DUTs/IO/Base/EtcSlaveTerminalBase_947E5A46.TcDUT

{attribute clr[Container(Layout.Stack)]}
{attribute clr[Group(Layout.GroupBox)]}
{attribute addProperty PreviousPort "Unknown"}
TYPE EtcSlaveTerminalBase_947E5A46 EXTENDS EtcSlaveBase_82538BE2 :
STRUCT
END_STRUCT
END_TYPE

// ---- DUTs/IO/Base/EtcSlaveBoxBase_77A0E4A7.TcDUT

{attribute clr[Container(Layout.Stack)]}
{attribute clr[Group(Layout.GroupBox)]}
{attribute addProperty PreviousPort "Unknown"}
TYPE EtcSlaveBoxBase_77A0E4A7 EXTENDS EtcSlaveBase_82538BE2 :
STRUCT
END_STRUCT
END_TYPE

// ---- DUTs/IO/Base/EtcSlaveEndTerminalBase_866C7F0C.TcDUT

{attribute clr[Container(Layout.Stack)]}
{attribute clr[Group(Layout.GroupBox)]}
{attribute addProperty PreviousPort "Unknown"}
TYPE EtcSlaveEndTerminalBase_866C7F0C EXTENDS EtcSlaveBase_82538BE2 :
STRUCT
END_STRUCT
END_TYPE

// ---- DUTs/IO/Base/InputBase_8311D824.TcDUT

TYPE InputBase_8311D824 :
STRUCT
END_STRUCT
END_TYPE

// ---- DUTs/IO/Base/OutputBase_10CEE7DE.TcDUT

